LIN {X 0,Y 292.683,Z 375.418,A -85,B 0,C 180,E1 -16601.198,E2 -16601.198} C_VEL
LIN {X 0,Y 293.911,Z 381.437,A -85,B 0,C 180,E1 -16604.861,E2 -16604.861} C_VEL
LIN {X 0,Y 294.978,Z 387.221,A -85,B 0,C 180,E1 -16608.157,E2 -16608.157} C_VEL
LIN {X 0,Y 295.925,Z 392.366,A -85,B 0,C 180,E1 -16610.924,E2 -16610.924} C_VEL
LIN {X 0,Y 296.024,Z 394.252,A -85,B 0,C 180,E1 -16611.884,E2 -16611.884} C_VEL
LIN {X 0,Y 294.406,Z 402.717,A -85,B 0,C 180,E1 -16615.877,E2 -16615.877} C_VEL
LIN {X 0,Y 292.727,Z 412.806,A -85,B 0,C 180,E1 -16620.517,E2 -16620.517} C_VEL
LIN {X 0,Y 291.994,Z 418.301,A -85,B 0,C 180,E1 -16622.943,E2 -16622.943} C_VEL
LIN {X 0,Y 294.998,Z 432.417,A -85,B 0,C 180,E1 -16623.88,E2 -16623.88} C_VEL
LIN {X 0,Y 296.907,Z 445.168,A -85,B 0,C 180,E1 -16624.923,E2 -16624.923} C_VEL
LIN {X 0,Y 297.945,Z 457.115,A -85,B 0,C 180,E1 -16626.095,E2 -16626.095} C_VEL
LIN {X 0,Y 298.202,Z 467.604,A -85,B 0,C 180,E1 -16627.301,E2 -16627.301} C_VEL
LIN {X 0,Y 297.752,Z 476.948,A -85,B 0,C 180,E1 -16628.541,E2 -16628.541} C_VEL
LIN {X 0,Y 296.927,Z 484.846,A -85,B 0,C 180,E1 -16629.748,E2 -16629.748} C_VEL
LIN {X 0,Y 294.74,Z 495.018,A -85,B 0,C 180,E1 -16631.583,E2 -16631.583} C_VEL
LIN {X 0,Y 292.887,Z 504.329,A -85,B 0,C 180,E1 -16633.704,E2 -16633.704} C_VEL
LIN {X 0,Y 291.885,Z 510.195,A -85,B 0,C 180,E1 -16635.357,E2 -16635.357} C_VEL
LIN {X 0,Y 290.834,Z 516.302,A -85,B 0,C 180,E1 -16637.44,E2 -16637.44} C_VEL
LIN {X 0,Y 290.21,Z 521.185,A -85,B 0,C 180,E1 -16639.536,E2 -16639.536} C_VEL
LIN {X 0,Y 290.014,Z 524.981,A -85,B 0,C 180,E1 -16641.641,E2 -16641.641} C_VEL
LIN {X 0,Y 290.054,Z 527.419,A -85,B 0,C 180,E1 -16643.428,E2 -16643.428} C_VEL
LIN {X 0,Y 290.356,Z 529.624,A -85,B 0,C 180,E1 -16645.837,E2 -16645.837} C_VEL
LIN {X 0,Y 290.572,Z 530.346,A -85,B 0,C 180,E1 -16647.228,E2 -16647.228} C_VEL
LIN {X 0,Y 290.579,Z 530.64,A -85,B 0,C 180,E1 -16648.615,E2 -16648.615} C_VEL
LIN {X 0,Y 290.692,Z 530.5,A -85,B 0,C 180,E1 -16650.001,E2 -16650.001} C_VEL
LIN {X 0,Y 290.641,Z 529.922,A -85,B 0,C 180,E1 -16651.387,E2 -16651.387} C_VEL
LIN {X 0,Y 290.644,Z 528.943,A -85,B 0,C 180,E1 -16652.773,E2 -16652.773} C_VEL
LIN {X 0,Y 290.521,Z 527.528,A -85,B 0,C 180,E1 -16654.163,E2 -16654.163} C_VEL
LIN {X 0,Y 290.267,Z 524.115,A -85,B 0,C 180,E1 -16656.483,E2 -16656.483} C_VEL
LIN {X 0,Y 290.179,Z 518.756,A -85,B 0,C 180,E1 -16659.059,E2 -16659.059} C_VEL
LIN {X 0,Y 290.446,Z 513.057,A -85,B 0,C 180,E1 -16661.163,E2 -16661.163} C_VEL
LIN {X 0,Y 291.073,Z 505.963,A -85,B 0,C 180,E1 -16663.262,E2 -16663.262} C_VEL
LIN {X 0,Y 291.825,Z 498.722,A -85,B 0,C 180,E1 -16665.005,E2 -16665.005} C_VEL
LIN {X 0,Y 293.098,Z 490.037,A -85,B 0,C 180,E1 -16666.724,E2 -16666.724} C_VEL
LIN {X 0,Y 294.416,Z 479.281,A -85,B 0,C 180,E1 -16668.44,E2 -16668.44} C_VEL
LIN {X 0,Y 294.522,Z 468.382,A -85,B 0,C 180,E1 -16669.88,E2 -16669.88} C_VEL
LIN {X 0,Y 294.174,Z 456.178,A -85,B 0,C 180,E1 -16671.185,E2 -16671.185} C_VEL
LIN {X 0,Y 293.492,Z 443.337,A -85,B 0,C 180,E1 -16672.251,E2 -16672.251} C_VEL
LIN {X 0,Y 292.3,Z 430.929,A -85,B 0,C 180,E1 -16673.044,E2 -16673.044} C_VEL
LIN {X 0,Y 290.807,Z 419.868,A -85,B 0,C 180,E1 -16673.595,E2 -16673.595} C_VEL
LIN {X 0,Y 291.778,Z 409.748,A -85,B 0,C 180,E1 -16678.015,E2 -16678.015} C_VEL
LIN {X 0,Y 292.997,Z 399.803,A -85,B 0,C 180,E1 -16682.41,E2 -16682.41} C_VEL
LIN {X 0,Y 294.364,Z 390.354,A -85,B 0,C 180,E1 -16686.648,E2 -16686.648} C_VEL
LIN {X 0,Y 294.622,Z 386.771,A -85,B 0,C 180,E1 -16688.333,E2 -16688.333} C_VEL
LIN {X 0,Y 293.697,Z 381.163,A -85,B 0,C 180,E1 -16691.126,E2 -16691.126} C_VEL
LIN {X 0,Y 292.259,Z 373.892,A -85,B 0,C 180,E1 -16694.951,E2 -16694.951} C_VEL
LIN {X 0,Y 291.394,Z 369.189,A -85,B 0,C 180,E1 -16697.647,E2 -16697.647} C_VEL
LIN {X 0,Y 291.357,Z 369.195,A -85,B 0,C 180,E1 -16701.159,E2 -16701.159} C_VEL
LIN {X 0,Y 291.365,Z 369.194,A -85,B 0,C 180,E1 -16704.627,E2 -16704.627} C_VEL
LIN {X 0,Y 291.375,Z 369.189,A -85,B 0,C 180,E1 -16707.951,E2 -16707.951} C_VEL
LIN {X 0,Y 291.382,Z 369.189,A -85,B 0,C 180,E1 -16711.158,E2 -16711.158} C_VEL
LIN {X 0,Y 291.417,Z 369.185,A -85,B 0,C 180,E1 -16714.272,E2 -16714.272} C_VEL
LIN {X 0,Y 291.387,Z 369.188,A -85,B 0,C 180,E1 -16717.3,E2 -16717.3} C_VEL
LIN {X 0,Y 291.463,Z 369.181,A -85,B 0,C 180,E1 -16720.271,E2 -16720.271} C_VEL
LIN {X 0,Y 291.56,Z 369.169,A -85,B 0,C 180,E1 -16724.624,E2 -16724.624} C_VEL
LIN {X 0,Y 291.542,Z 369.169,A -85,B 0,C 180,E1 -16728.881,E2 -16728.881} C_VEL
LIN {X 0,Y 291.716,Z 369.146,A -85,B 0,C 180,E1 -16731.689,E2 -16731.689} C_VEL
LIN {X 0,Y 291.636,Z 369.159,A -85,B 0,C 180,E1 -16734.469,E2 -16734.469} C_VEL
LIN {X 0,Y 291.895,Z 369.121,A -85,B 0,C 180,E1 -16738.621,E2 -16738.621} C_VEL
LIN {X 0,Y 291.896,Z 369.122,A -85,B 0,C 180,E1 -16741.38,E2 -16741.38} C_VEL
LIN {X 0,Y 291.753,Z 369.136,A -85,B 0,C 180,E1 -16746.918,E2 -16746.918} C_VEL
LIN {X 0,Y 291.635,Z 369.156,A -85,B 0,C 180,E1 -16749.712,E2 -16749.712} C_VEL
LIN {X 0,Y 291.528,Z 369.169,A -85,B 0,C 180,E1 -16753.95,E2 -16753.95} C_VEL
LIN {X 0,Y 291.493,Z 369.171,A -85,B 0,C 180,E1 -16756.818,E2 -16756.818} C_VEL
LIN {X 0,Y 291.457,Z 369.181,A -85,B 0,C 180,E1 -16759.875,E2 -16759.875} C_VEL
LIN {X 0,Y 291.407,Z 369.184,A -85,B 0,C 180,E1 -16764.205,E2 -16764.205} C_VEL
LIN {X 0,Y 291.427,Z 369.183,A -85,B 0,C 180,E1 -16767.272,E2 -16767.272} C_VEL
LIN {X 0,Y 291.343,Z 369.188,A -85,B 0,C 180,E1 -16770.437,E2 -16770.437} C_VEL
LIN {X 0,Y 291.351,Z 369.194,A -85,B 0,C 180,E1 -16773.698,E2 -16773.698} C_VEL
LIN {X 0,Y 291.401,Z 369.187,A -85,B 0,C 180,E1 -16777.259,E2 -16777.259} C_VEL
LIN {X 0,Y 291.341,Z 369.192,A -85,B 0,C 180,E1 -16780.642,E2 -16780.642} C_VEL
LIN {X 0,Y 291.32,Z 369.193,A -85,B 0,C 180,E1 -16784.397,E2 -16784.397} C_VEL
LIN {X 0,Y 291.333,Z 369.192,A -85,B 0,C 180,E1 -16788.404,E2 -16788.404} C_VEL
LIN {X 0,Y 291.359,Z 369.193,A -85,B 0,C 180,E1 -16791.158,E2 -16791.158} C_VEL
LIN {X 0,Y 291.367,Z 369.189,A -85,B 0,C 180,E1 -16794.626,E2 -16794.626} C_VEL
LIN {X 0,Y 291.378,Z 369.187,A -85,B 0,C 180,E1 -16797.95,E2 -16797.95} C_VEL
LIN {X 0,Y 291.389,Z 369.19,A -85,B 0,C 180,E1 -16801.158,E2 -16801.158} C_VEL
LIN {X 0,Y 291.423,Z 369.183,A -85,B 0,C 180,E1 -16804.271,E2 -16804.271} C_VEL
LIN {X 0,Y 291.388,Z 369.189,A -85,B 0,C 180,E1 -16807.299,E2 -16807.299} C_VEL
LIN {X 0,Y 291.464,Z 369.178,A -85,B 0,C 180,E1 -16810.27,E2 -16810.27} C_VEL
LIN {X 0,Y 291.563,Z 369.169,A -85,B 0,C 180,E1 -16814.837,E2 -16814.837} C_VEL
LIN {X 0,Y 291.568,Z 369.167,A -85,B 0,C 180,E1 -16815.316,E2 -16815.316} C_VEL
LIN {X 0,Y 295.833,Z 381.993,A -85,B 0,C 180,E1 -16816.562,E2 -16816.562} C_VEL
LIN {X 0,Y 298.818,Z 392.412,A -85,B 0,C 180,E1 -16817.779,E2 -16817.779} C_VEL
LIN {X 0,Y 299.175,Z 393.845,A -85,B 0,C 180,E1 -16817.965,E2 -16817.965} C_VEL
LIN {X 0,Y 298.005,Z 405.109,A -85,B 0,C 180,E1 -16819.296,E2 -16819.296} C_VEL
LIN {X 0,Y 296.886,Z 415.247,A -85,B 0,C 180,E1 -16820.804,E2 -16820.804} C_VEL
LIN {X 0,Y 295.741,Z 424.376,A -85,B 0,C 180,E1 -16822.489,E2 -16822.489} C_VEL
LIN {X 0,Y 294.418,Z 433.245,A -85,B 0,C 180,E1 -16824.52,E2 -16824.52} C_VEL
LIN {X 0,Y 293.334,Z 440.396,A -85,B 0,C 180,E1 -16826.565,E2 -16826.565} C_VEL
LIN {X 0,Y 292.496,Z 446.124,A -85,B 0,C 180,E1 -16828.622,E2 -16828.622} C_VEL
LIN {X 0,Y 291.905,Z 450.636,A -85,B 0,C 180,E1 -16830.689,E2 -16830.689} C_VEL
LIN {X 0,Y 291.33,Z 454.107,A -85,B 0,C 180,E1 -16832.764,E2 -16832.764} C_VEL
LIN {X 0,Y 291.196,Z 455.839,A -85,B 0,C 180,E1 -16834.151,E2 -16834.151} C_VEL
LIN {X 0,Y 291.213,Z 457.151,A -85,B 0,C 180,E1 -16835.539,E2 -16835.539} C_VEL
LIN {X 0,Y 291.178,Z 458.652,A -85,B 0,C 180,E1 -16838.269,E2 -16838.269} C_VEL
LIN {X 0,Y 291.268,Z 458.81,A -85,B 0,C 180,E1 -16839.723,E2 -16839.723} C_VEL
LIN {X 0,Y 291.675,Z 457.948,A -85,B 0,C 180,E1 -16842.523,E2 -16842.523} C_VEL
LIN {X 0,Y 292.039,Z 456.928,A -85,B 0,C 180,E1 -16843.924,E2 -16843.924} C_VEL
LIN {X 0,Y 292.98,Z 454.095,A -85,B 0,C 180,E1 -16846.356,E2 -16846.356} C_VEL
LIN {X 0,Y 294.179,Z 449.853,A -85,B 0,C 180,E1 -16848.814,E2 -16848.814} C_VEL
LIN {X 0,Y 295.431,Z 445.004,A -85,B 0,C 180,E1 -16850.905,E2 -16850.905} C_VEL
LIN {X 0,Y 296.905,Z 439.068,A -85,B 0,C 180,E1 -16852.915,E2 -16852.915} C_VEL
LIN {X 0,Y 298.493,Z 432.492,A -85,B 0,C 180,E1 -16854.702,E2 -16854.702} C_VEL
LIN {X 0,Y 300.367,Z 423.575,A -85,B 0,C 180,E1 -16856.659,E2 -16856.659} C_VEL
LIN {X 0,Y 302.222,Z 413.214,A -85,B 0,C 180,E1 -16858.47,E2 -16858.47} C_VEL
LIN {X 0,Y 303.808,Z 403.47,A -85,B 0,C 180,E1 -16859.825,E2 -16859.825} C_VEL
LIN {X 0,Y 303.684,Z 401.365,A -85,B 0,C 180,E1 -16860.122,E2 -16860.122} C_VEL
LIN {X 0,Y 300.573,Z 391.397,A -85,B 0,C 180,E1 -16861.672,E2 -16861.672} C_VEL
LIN {X 0,Y 296.215,Z 380.226,A -85,B 0,C 180,E1 -16863.243,E2 -16863.243} C_VEL
LIN {X 0,Y 292.253,Z 371.834,A -85,B 0,C 180,E1 -16864.331,E2 -16864.331} C_VEL
LIN {X 0,Y 291.371,Z 369.192,A -85,B 0,C 180,E1 -16864.659,E2 -16864.659} C_VEL
LIN {X 0,Y 291.376,Z 369.194,A -85,B 0,C 180,E1 -16867.253,E2 -16867.253} C_VEL
LIN {X 0,Y 291.332,Z 369.197,A -85,B 0,C 180,E1 -16870.641,E2 -16870.641} C_VEL
LIN {X 0,Y 291.288,Z 369.2,A -85,B 0,C 180,E1 -16874.401,E2 -16874.401} C_VEL
LIN {X 0,Y 291.354,Z 369.197,A -85,B 0,C 180,E1 -16878.397,E2 -16878.397} C_VEL
LIN {X 0,Y 291.379,Z 369.192,A -85,B 0,C 180,E1 -16881.162,E2 -16881.162} C_VEL
LIN {X 0,Y 291.384,Z 369.188,A -85,B 0,C 180,E1 -16884.629,E2 -16884.629} C_VEL
LIN {X 0,Y 291.373,Z 369.173,A -85,B 0,C 180,E1 -16887.95,E2 -16887.95} C_VEL
LIN {X 0,Y 291.38,Z 369.158,A -85,B 0,C 180,E1 -16891.158,E2 -16891.158} C_VEL
LIN {X 0,Y 291.414,Z 369.185,A -85,B 0,C 180,E1 -16894.271,E2 -16894.271} C_VEL
LIN {X 0,Y 291.379,Z 369.178,A -85,B 0,C 180,E1 -16897.299,E2 -16897.299} C_VEL
LIN {X 0,Y 291.455,Z 369.179,A -85,B 0,C 180,E1 -16900.27,E2 -16900.27} C_VEL
LIN {X 0,Y 291.551,Z 369.17,A -85,B 0,C 180,E1 -16904.623,E2 -16904.623} C_VEL
LIN {X 0,Y 291.535,Z 369.171,A -85,B 0,C 180,E1 -16908.88,E2 -16908.88} C_VEL
LIN {X 0,Y 291.705,Z 369.15,A -85,B 0,C 180,E1 -16911.688,E2 -16911.688} C_VEL
LIN {X 0,Y 291.603,Z 369.148,A -85,B 0,C 180,E1 -16914.707,E2 -16914.707} C_VEL
LIN {X 0,Y 291.89,Z 369.123,A -85,B 0,C 180,E1 -16918.62,E2 -16918.62} C_VEL
LIN {X 0,Y 291.91,Z 369.114,A -85,B 0,C 180,E1 -16920.74,E2 -16920.74} C_VEL
LIN {X 0,Y 291.165,Z 369.216,A -85,B 0,C 180,E1 -16921.888,E2 -16921.888} C_VEL
LIN {X 0,Y 288.167,Z 369.588,A -85,B 0,C 180,E1 -16923.754,E2 -16923.754} C_VEL
LIN {X 0,Y 285.7,Z 369.889,A -85,B 0,C 180,E1 -16925.27,E2 -16925.27} C_VEL
LIN {X 0,Y 284.71,Z 370.017,A -85,B 0,C 180,E1 -16926.448,E2 -16926.448} C_VEL
LIN {X 0,Y 284.666,Z 370.023,A -85,B 0,C 180,E1 -16926.846,E2 -16926.846} C_VEL
LIN {X 0,Y 284.562,Z 370.029,A -85,B 0,C 180,E1 -16929.955,E2 -16929.955} C_VEL
LIN {X 0,Y 284.477,Z 370.042,A -85,B 0,C 180,E1 -16934.303,E2 -16934.303} C_VEL
LIN {X 0,Y 284.421,Z 370.051,A -85,B 0,C 180,E1 -16937.248,E2 -16937.248} C_VEL
LIN {X 0,Y 284.374,Z 370.06,A -85,B 0,C 180,E1 -16940.242,E2 -16940.242} C_VEL
LIN {X 0,Y 284.365,Z 370.061,A -85,B 0,C 180,E1 -16943.876,E2 -16943.876} C_VEL
LIN {X 0,Y 284.393,Z 370.064,A -85,B 0,C 180,E1 -16947.174,E2 -16947.174} C_VEL
LIN {X 0,Y 284.292,Z 370.076,A -85,B 0,C 180,E1 -16951.275,E2 -16951.275} C_VEL
LIN {X 0,Y 284.345,Z 370.064,A -85,B 0,C 180,E1 -16955.803,E2 -16955.803} C_VEL
LIN {X 0,Y 284.38,Z 370.218,A -85,B 0,C 180,E1 -16956.379,E2 -16956.379} C_VEL
LIN {X 0,Y 285.532,Z 375.84,A -85,B 0,C 180,E1 -16960.27,E2 -16960.27} C_VEL
LIN {X 0,Y 286.736,Z 381.797,A -85,B 0,C 180,E1 -16964.061,E2 -16964.061} C_VEL
LIN {X 0,Y 288,Z 388.459,A -85,B 0,C 180,E1 -16967.97,E2 -16967.97} C_VEL
LIN {X 0,Y 289,Z 394.136,A -85,B 0,C 180,E1 -16971.095,E2 -16971.095} C_VEL
LIN {X 0,Y 288.762,Z 396.965,A -85,B 0,C 180,E1 -16972.523,E2 -16972.523} C_VEL
LIN {X 0,Y 286.964,Z 405.919,A -85,B 0,C 180,E1 -16976.845,E2 -16976.845} C_VEL
LIN {X 0,Y 285.399,Z 415.403,A -85,B 0,C 180,E1 -16981.303,E2 -16981.303} C_VEL
LIN {X 0,Y 285.143,Z 417.2,A -85,B 0,C 180,E1 -16982.13,E2 -16982.13} C_VEL
LIN {X 0,Y 287.856,Z 429.507,A -85,B 0,C 180,E1 -16982.975,E2 -16982.975} C_VEL
LIN {X 0,Y 289.99,Z 442.581,A -85,B 0,C 180,E1 -16984.06,E2 -16984.06} C_VEL
LIN {X 0,Y 291.121,Z 454.499,A -85,B 0,C 180,E1 -16985.231,E2 -16985.231} C_VEL
LIN {X 0,Y 291.522,Z 466.194,A -85,B 0,C 180,E1 -16986.6,E2 -16986.6} C_VEL
LIN {X 0,Y 291.067,Z 476.581,A -85,B 0,C 180,E1 -16988.023,E2 -16988.023} C_VEL
LIN {X 0,Y 290.038,Z 485.402,A -85,B 0,C 180,E1 -16989.431,E2 -16989.431} C_VEL
LIN {X 0,Y 287.993,Z 494.494,A -85,B 0,C 180,E1 -16991.136,E2 -16991.136} C_VEL
LIN {X 0,Y 286.038,Z 503.818,A -85,B 0,C 180,E1 -16993.324,E2 -16993.324} C_VEL
LIN {X 0,Y 284.721,Z 510.666,A -85,B 0,C 180,E1 -16995.345,E2 -16995.345} C_VEL
LIN {X 0,Y 283.581,Z 517.334,A -85,B 0,C 180,E1 -16997.84,E2 -16997.84} C_VEL
LIN {X 0,Y 283.059,Z 521.803,A -85,B 0,C 180,E1 -16999.992,E2 -16999.992} C_VEL
LIN {X 0,Y 282.934,Z 524.207,A -85,B 0,C 180,E1 -17001.43,E2 -17001.43} C_VEL
LIN {X 0,Y 282.99,Z 526.775,A -85,B 0,C 180,E1 -17003.409,E2 -17003.409} C_VEL
LIN {X 0,Y 283.275,Z 528.786,A -85,B 0,C 180,E1 -17005.733,E2 -17005.733} C_VEL
LIN {X 0,Y 283.52,Z 529.496,A -85,B 0,C 180,E1 -17007.159,E2 -17007.159} C_VEL
LIN {X 0,Y 283.531,Z 529.768,A -85,B 0,C 180,E1 -17008.581,E2 -17008.581} C_VEL
LIN {X 0,Y 283.647,Z 529.602,A -85,B 0,C 180,E1 -17010.001,E2 -17010.001} C_VEL
LIN {X 0,Y 283.593,Z 529.007,A -85,B 0,C 180,E1 -17011.421,E2 -17011.421} C_VEL
LIN {X 0,Y 283.596,Z 528.01,A -85,B 0,C 180,E1 -17012.842,E2 -17012.842} C_VEL
LIN {X 0,Y 283.455,Z 526.566,A -85,B 0,C 180,E1 -17014.267,E2 -17014.267} C_VEL
LIN {X 0,Y 283.181,Z 522.613,A -85,B 0,C 180,E1 -17016.917,E2 -17016.917} C_VEL
LIN {X 0,Y 283.108,Z 517.697,A -85,B 0,C 180,E1 -17019.287,E2 -17019.287} C_VEL
LIN {X 0,Y 283.414,Z 511.954,A -85,B 0,C 180,E1 -17021.443,E2 -17021.443} C_VEL
LIN {X 0,Y 284.098,Z 504.802,A -85,B 0,C 180,E1 -17023.593,E2 -17023.593} C_VEL
LIN {X 0,Y 284.849,Z 497.495,A -85,B 0,C 180,E1 -17025.382,E2 -17025.382} C_VEL
LIN {X 0,Y 286.409,Z 487.741,A -85,B 0,C 180,E1 -17027.31,E2 -17027.31} C_VEL
LIN {X 0,Y 287.492,Z 477.857,A -85,B 0,C 180,E1 -17028.9,E2 -17028.9} C_VEL
LIN {X 0,Y 287.492,Z 466.799,A -85,B 0,C 180,E1 -17030.388,E2 -17030.388} C_VEL
LIN {X 0,Y 287.242,Z 454.552,A -85,B 0,C 180,E1 -17031.702,E2 -17031.702} C_VEL
LIN {X 0,Y 286.492,Z 441.166,A -85,B 0,C 180,E1 -17032.825,E2 -17032.825} C_VEL
LIN {X 0,Y 285.104,Z 428.095,A -85,B 0,C 180,E1 -17033.66,E2 -17033.66} C_VEL
LIN {X 0,Y 283.82,Z 419.071,A -85,B 0,C 180,E1 -17034.101,E2 -17034.101} C_VEL
LIN {X 0,Y 284.864,Z 408.71,A -85,B 0,C 180,E1 -17038.758,E2 -17038.758} C_VEL
LIN {X 0,Y 286.02,Z 399.96,A -85,B 0,C 180,E1 -17042.724,E2 -17042.724} C_VEL
LIN {X 0,Y 287.363,Z 391.118,A -85,B 0,C 180,E1 -17046.82,E2 -17046.82} C_VEL
LIN {X 0,Y 287.573,Z 387.519,A -85,B 0,C 180,E1 -17048.551,E2 -17048.551} C_VEL
LIN {X 0,Y 286.398,Z 380.811,A -85,B 0,C 180,E1 -17052.007,E2 -17052.007} C_VEL
LIN {X 0,Y 284.901,Z 372.942,A -85,B 0,C 180,E1 -17056.314,E2 -17056.314} C_VEL
LIN {X 0,Y 284.329,Z 370.069,A -85,B 0,C 180,E1 -17058.057,E2 -17058.057} C_VEL
LIN {X 0,Y 284.326,Z 370.069,A -85,B 0,C 180,E1 -17062.279,E2 -17062.279} C_VEL
LIN {X 0,Y 284.313,Z 370.071,A -85,B 0,C 180,E1 -17065.351,E2 -17065.351} C_VEL
LIN {X 0,Y 284.298,Z 370.073,A -85,B 0,C 180,E1 -17068.726,E2 -17068.726} C_VEL
LIN {X 0,Y 284.399,Z 370.061,A -85,B 0,C 180,E1 -17072.828,E2 -17072.828} C_VEL
LIN {X 0,Y 284.372,Z 370.066,A -85,B 0,C 180,E1 -17076.708,E2 -17076.708} C_VEL
LIN {X 0,Y 284.409,Z 370.058,A -85,B 0,C 180,E1 -17081.262,E2 -17081.262} C_VEL
LIN {X 0,Y 284.498,Z 370.05,A -85,B 0,C 180,E1 -17084.46,E2 -17084.46} C_VEL
LIN {X 0,Y 284.494,Z 370.049,A -85,B 0,C 180,E1 -17088.602,E2 -17088.602} C_VEL
LIN {X 0,Y 284.666,Z 370.024,A -85,B 0,C 180,E1 -17091.482,E2 -17091.482} C_VEL
LIN {X 0,Y 284.607,Z 370.036,A -85,B 0,C 180,E1 -17094.332,E2 -17094.332} C_VEL
LIN {X 0,Y 284.861,Z 369.997,A -85,B 0,C 180,E1 -17098.587,E2 -17098.587} C_VEL
LIN {X 0,Y 284.862,Z 369.998,A -85,B 0,C 180,E1 -17101.414,E2 -17101.414} C_VEL
LIN {X 0,Y 284.705,Z 370.013,A -85,B 0,C 180,E1 -17107.09,E2 -17107.09} C_VEL
LIN {X 0,Y 284.573,Z 370.038,A -85,B 0,C 180,E1 -17109.956,E2 -17109.956} C_VEL
LIN {X 0,Y 284.488,Z 370.042,A -85,B 0,C 180,E1 -17114.303,E2 -17114.303} C_VEL
LIN {X 0,Y 284.432,Z 370.051,A -85,B 0,C 180,E1 -17117.248,E2 -17117.248} C_VEL
LIN {X 0,Y 284.386,Z 370.059,A -85,B 0,C 180,E1 -17120.242,E2 -17120.242} C_VEL
LIN {X 0,Y 284.376,Z 370.06,A -85,B 0,C 180,E1 -17123.875,E2 -17123.875} C_VEL
LIN {X 0,Y 284.402,Z 370.057,A -85,B 0,C 180,E1 -17127.173,E2 -17127.173} C_VEL
LIN {X 0,Y 284.302,Z 370.067,A -85,B 0,C 180,E1 -17131.274,E2 -17131.274} C_VEL
LIN {X 0,Y 284.368,Z 370.064,A -85,B 0,C 180,E1 -17135.354,E2 -17135.354} C_VEL
LIN {X 0,Y 284.329,Z 370.065,A -85,B 0,C 180,E1 -17138.167,E2 -17138.167} C_VEL
LIN {X 0,Y 284.275,Z 370.071,A -85,B 0,C 180,E1 -17142.124,E2 -17142.124} C_VEL
LIN {X 0,Y 284.274,Z 370.071,A -85,B 0,C 180,E1 -17146.192,E2 -17146.192} C_VEL
LIN {X 0,Y 284.312,Z 370.066,A -85,B 0,C 180,E1 -17150.024,E2 -17150.024} C_VEL
LIN {X 0,Y 284.338,Z 370.065,A -85,B 0,C 180,E1 -17153.614,E2 -17153.614} C_VEL
LIN {X 0,Y 284.314,Z 370.071,A -85,B 0,C 180,E1 -17157.189,E2 -17157.189} C_VEL
LIN {X 0,Y 284.365,Z 370.062,A -85,B 0,C 180,E1 -17160.376,E2 -17160.376} C_VEL
LIN {X 0,Y 284.384,Z 370.06,A -85,B 0,C 180,E1 -17163.586,E2 -17163.586} C_VEL
LIN {X 0,Y 284.373,Z 370.063,A -85,B 0,C 180,E1 -17166.706,E2 -17166.706} C_VEL
LIN {X 0,Y 284.41,Z 370.059,A -85,B 0,C 180,E1 -17171.261,E2 -17171.261} C_VEL
LIN {X 0,Y 284.543,Z 370.186,A -85,B 0,C 180,E1 -17174.821,E2 -17174.821} C_VEL
LIN {X 0,Y 288.815,Z 382.8,A -85,B 0,C 180,E1 -17176.09,E2 -17176.09} C_VEL
LIN {X 0,Y 291.742,Z 392.861,A -85,B 0,C 180,E1 -17177.3,E2 -17177.3} C_VEL
LIN {X 0,Y 292.372,Z 395.773,A -85,B 0,C 180,E1 -17177.681,E2 -17177.681} C_VEL
LIN {X 0,Y 291.132,Z 406.849,A -85,B 0,C 180,E1 -17179.04,E2 -17179.04} C_VEL
LIN {X 0,Y 289.982,Z 416.81,A -85,B 0,C 180,E1 -17180.583,E2 -17180.583} C_VEL
LIN {X 0,Y 288.793,Z 425.792,A -85,B 0,C 180,E1 -17182.307,E2 -17182.307} C_VEL
LIN {X 0,Y 287.426,Z 434.571,A -85,B 0,C 180,E1 -17184.386,E2 -17184.386} C_VEL
LIN {X 0,Y 286.316,Z 441.641,A -85,B 0,C 180,E1 -17186.481,E2 -17186.481} C_VEL
LIN {X 0,Y 285.463,Z 447.282,A -85,B 0,C 180,E1 -17188.588,E2 -17188.588} C_VEL
LIN {X 0,Y 284.859,Z 451.727,A -85,B 0,C 180,E1 -17190.706,E2 -17190.706} C_VEL
LIN {X 0,Y 284.272,Z 455.146,A -85,B 0,C 180,E1 -17192.833,E2 -17192.833} C_VEL
LIN {X 0,Y 284.157,Z 458.121,A -85,B 0,C 180,E1 -17195.677,E2 -17195.677} C_VEL
LIN {X 0,Y 284.146,Z 459.529,A -85,B 0,C 180,E1 -17198.365,E2 -17198.365} C_VEL
LIN {X 0,Y 284.256,Z 459.674,A -85,B 0,C 180,E1 -17199.965,E2 -17199.965} C_VEL
LIN {X 0,Y 284.715,Z 458.759,A -85,B 0,C 180,E1 -17202.835,E2 -17202.835} C_VEL
LIN {X 0,Y 285.109,Z 457.687,A -85,B 0,C 180,E1 -17204.27,E2 -17204.27} C_VEL
LIN {X 0,Y 286.057,Z 454.984,A -85,B 0,C 180,E1 -17206.628,E2 -17206.628} C_VEL
LIN {X 0,Y 287.401,Z 450.491,A -85,B 0,C 180,E1 -17209.275,E2 -17209.275} C_VEL
LIN {X 0,Y 288.743,Z 445.575,A -85,B 0,C 180,E1 -17211.413,E2 -17211.413} C_VEL
LIN {X 0,Y 290.322,Z 439.561,A -85,B 0,C 180,E1 -17213.466,E2 -17213.466} C_VEL
LIN {X 0,Y 292.307,Z 431.428,A -85,B 0,C 180,E1 -17215.643,E2 -17215.643} C_VEL
LIN {X 0,Y 294.169,Z 422.87,A -85,B 0,C 180,E1 -17217.476,E2 -17217.476} C_VEL
LIN {X 0,Y 295.925,Z 413.351,A -85,B 0,C 180,E1 -17219.133,E2 -17219.133} C_VEL
LIN {X 0,Y 297.285,Z 405.45,A -85,B 0,C 180,E1 -17220.247,E2 -17220.247} C_VEL
LIN {X 0,Y 297.101,Z 402.931,A -85,B 0,C 180,E1 -17220.631,E2 -17220.631} C_VEL
LIN {X 0,Y 293.658,Z 392.367,A -85,B 0,C 180,E1 -17222.355,E2 -17222.355} C_VEL
LIN {X 0,Y 289.363,Z 381.424,A -85,B 0,C 180,E1 -17223.959,E2 -17223.959} C_VEL
LIN {X 0,Y 285.305,Z 372.882,A -85,B 0,C 180,E1 -17225.12,E2 -17225.12} C_VEL
LIN {X 0,Y 284.331,Z 370.073,A -85,B 0,C 180,E1 -17225.456,E2 -17225.456} C_VEL
LIN {X 0,Y 284.312,Z 370.07,A -85,B 0,C 180,E1 -17228.168,E2 -17228.168} C_VEL
LIN {X 0,Y 284.268,Z 370.074,A -85,B 0,C 180,E1 -17232.123,E2 -17232.123} C_VEL
LIN {X 0,Y 284.271,Z 370.077,A -85,B 0,C 180,E1 -17236.191,E2 -17236.191} C_VEL
LIN {X 0,Y 284.35,Z 370.063,A -85,B 0,C 180,E1 -17240.012,E2 -17240.012} C_VEL
LIN {X 0,Y 284.353,Z 370.06,A -85,B 0,C 180,E1 -17243.617,E2 -17243.617} C_VEL
LIN {X 0,Y 284.307,Z 370.063,A -85,B 0,C 180,E1 -17247.188,E2 -17247.188} C_VEL
LIN {X 0,Y 284.357,Z 370.025,A -85,B 0,C 180,E1 -17250.375,E2 -17250.375} C_VEL
LIN {X 0,Y 284.375,Z 370.059,A -85,B 0,C 180,E1 -17253.586,E2 -17253.586} C_VEL
LIN {X 0,Y 284.363,Z 370.051,A -85,B 0,C 180,E1 -17256.706,E2 -17256.706} C_VEL
LIN {X 0,Y 284.401,Z 370.052,A -85,B 0,C 180,E1 -17261.261,E2 -17261.261} C_VEL
LIN {X 0,Y 284.489,Z 370.049,A -85,B 0,C 180,E1 -17264.458,E2 -17264.458} C_VEL
LIN {X 0,Y 284.487,Z 370.049,A -85,B 0,C 180,E1 -17268.601,E2 -17268.601} C_VEL
LIN {X 0,Y 284.656,Z 370.028,A -85,B 0,C 180,E1 -17271.481,E2 -17271.481} C_VEL
LIN {X 0,Y 284.599,Z 370.02,A -85,B 0,C 180,E1 -17274.331,E2 -17274.331} C_VEL
LIN {X 0,Y 284.856,Z 369.999,A -85,B 0,C 180,E1 -17278.586,E2 -17278.586} C_VEL
LIN {X 0,Y 284.856,Z 369.999,A -85,B 0,C 180,E1 -17281.413,E2 -17281.413} C_VEL
LIN {X 0,Y 284.666,Z 370.023,A -85,B 0,C 180,E1 -17286.846,E2 -17286.846} C_VEL
LIN {X 0,Y 284.057,Z 370.107,A -85,B 0,C 180,E1 -17288.026,E2 -17288.026} C_VEL
LIN {X 0,Y 281.098,Z 370.474,A -85,B 0,C 180,E1 -17289.942,E2 -17289.942} C_VEL
LIN {X 0,Y 278.55,Z 370.787,A -85,B 0,C 180,E1 -17291.5,E2 -17291.5} C_VEL
LIN {X 0,Y 277.48,Z 370.92,A -85,B 0,C 180,E1 -17292.711,E2 -17292.711} C_VEL
LIN {X 0,Y 277.41,Z 370.924,A -85,B 0,C 180,E1 -17293.122,E2 -17293.122} C_VEL
LIN {X 0,Y 277.402,Z 370.931,A -85,B 0,C 180,E1 -17296.182,E2 -17296.182} C_VEL
LIN {X 0,Y 277.341,Z 370.935,A -85,B 0,C 180,E1 -17300.35,E2 -17300.35} C_VEL
LIN {X 0,Y 277.315,Z 370.94,A -85,B 0,C 180,E1 -17304.171,E2 -17304.171} C_VEL
LIN {X 0,Y 277.322,Z 370.945,A -85,B 0,C 180,E1 -17307.506,E2 -17307.506} C_VEL
LIN {X 0,Y 277.268,Z 370.951,A -85,B 0,C 180,E1 -17310.482,E2 -17310.482} C_VEL
LIN {X 0,Y 277.313,Z 370.941,A -85,B 0,C 180,E1 -17315.209,E2 -17315.209} C_VEL
LIN {X 0,Y 277.411,Z 371.459,A -85,B 0,C 180,E1 -17315.838,E2 -17315.838} C_VEL
LIN {X 0,Y 278.625,Z 377.319,A -85,B 0,C 180,E1 -17320.009,E2 -17320.009} C_VEL
LIN {X 0,Y 279.768,Z 383.119,A -85,B 0,C 180,E1 -17323.819,E2 -17323.819} C_VEL
LIN {X 0,Y 280.917,Z 389.221,A -85,B 0,C 180,E1 -17327.509,E2 -17327.509} C_VEL
LIN {X 0,Y 281.911,Z 394.639,A -85,B 0,C 180,E1 -17330.608,E2 -17330.608} C_VEL
LIN {X 0,Y 282.033,Z 396.233,A -85,B 0,C 180,E1 -17331.468,E2 -17331.468} C_VEL
LIN {X 0,Y 280.998,Z 401.291,A -85,B 0,C 180,E1 -17334.004,E2 -17334.004} C_VEL
LIN {X 0,Y 279.392,Z 409.647,A -85,B 0,C 180,E1 -17338.114,E2 -17338.114} C_VEL
LIN {X 0,Y 278.331,Z 416.232,A -85,B 0,C 180,E1 -17341.28,E2 -17341.28} C_VEL
LIN {X 0,Y 281.135,Z 429.112,A -85,B 0,C 180,E1 -17342.204,E2 -17342.204} C_VEL
LIN {X 0,Y 283.236,Z 441.536,A -85,B 0,C 180,E1 -17343.288,E2 -17343.288} C_VEL
LIN {X 0,Y 284.486,Z 454.58,A -85,B 0,C 180,E1 -17344.629,E2 -17344.629} C_VEL
LIN {X 0,Y 284.823,Z 466.832,A -85,B 0,C 180,E1 -17346.136,E2 -17346.136} C_VEL
LIN {X 0,Y 284.267,Z 477.4,A -85,B 0,C 180,E1 -17347.66,E2 -17347.66} C_VEL
LIN {X 0,Y 283.368,Z 484.949,A -85,B 0,C 180,E1 -17348.924,E2 -17348.924} C_VEL
LIN {X 0,Y 281.251,Z 493.969,A -85,B 0,C 180,E1 -17350.666,E2 -17350.666} C_VEL
LIN {X 0,Y 279.237,Z 503.019,A -85,B 0,C 180,E1 -17352.848,E2 -17352.848} C_VEL
LIN {X 0,Y 277.842,Z 510.005,A -85,B 0,C 180,E1 -17354.974,E2 -17354.974} C_VEL
LIN {X 0,Y 276.576,Z 516.623,A -85,B 0,C 180,E1 -17357.527,E2 -17357.527} C_VEL
LIN {X 0,Y 276.007,Z 521.052,A -85,B 0,C 180,E1 -17359.734,E2 -17359.734} C_VEL
LIN {X 0,Y 275.881,Z 523.439,A -85,B 0,C 180,E1 -17361.209,E2 -17361.209} C_VEL
LIN {X 0,Y 275.934,Z 526.118,A -85,B 0,C 180,E1 -17363.376,E2 -17363.376} C_VEL
LIN {X 0,Y 276.197,Z 527.95,A -85,B 0,C 180,E1 -17365.623,E2 -17365.623} C_VEL
LIN {X 0,Y 276.467,Z 528.647,A -85,B 0,C 180,E1 -17367.087,E2 -17367.087} C_VEL
LIN {X 0,Y 276.483,Z 528.889,A -85,B 0,C 180,E1 -17368.544,E2 -17368.544} C_VEL
LIN {X 0,Y 276.602,Z 528.704,A -85,B 0,C 180,E1 -17370.001,E2 -17370.001} C_VEL
LIN {X 0,Y 276.545,Z 528.092,A -85,B 0,C 180,E1 -17371.457,E2 -17371.457} C_VEL
LIN {X 0,Y 276.548,Z 527.077,A -85,B 0,C 180,E1 -17372.914,E2 -17372.914} C_VEL
LIN {X 0,Y 276.39,Z 525.597,A -85,B 0,C 180,E1 -17374.376,E2 -17374.376} C_VEL
LIN {X 0,Y 276.107,Z 521.893,A -85,B 0,C 180,E1 -17376.926,E2 -17376.926} C_VEL
LIN {X 0,Y 276.061,Z 516.639,A -85,B 0,C 180,E1 -17379.526,E2 -17379.526} C_VEL
LIN {X 0,Y 276.393,Z 510.847,A -85,B 0,C 180,E1 -17381.738,E2 -17381.738} C_VEL
LIN {X 0,Y 277.126,Z 503.622,A -85,B 0,C 180,E1 -17383.942,E2 -17383.942} C_VEL
LIN {X 0,Y 278.215,Z 494.596,A -85,B 0,C 180,E1 -17386.134,E2 -17386.134} C_VEL
LIN {X 0,Y 279.5,Z 486.404,A -85,B 0,C 180,E1 -17387.752,E2 -17387.752} C_VEL
LIN {X 0,Y 280.501,Z 477.629,A -85,B 0,C 180,E1 -17389.2,E2 -17389.2} C_VEL
LIN {X 0,Y 280.519,Z 466.905,A -85,B 0,C 180,E1 -17390.7,E2 -17390.7} C_VEL
LIN {X 0,Y 280.327,Z 454.561,A -85,B 0,C 180,E1 -17392.091,E2 -17392.091} C_VEL
LIN {X 0,Y 279.653,Z 441.73,A -85,B 0,C 180,E1 -17393.22,E2 -17393.22} C_VEL
LIN {X 0,Y 278.307,Z 428.481,A -85,B 0,C 180,E1 -17394.12,E2 -17394.12} C_VEL
LIN {X 0,Y 276.834,Z 418.137,A -85,B 0,C 180,E1 -17394.667,E2 -17394.667} C_VEL
LIN {X 0,Y 277.996,Z 407.628,A -85,B 0,C 180,E1 -17399.538,E2 -17399.538} C_VEL
LIN {X 0,Y 279.267,Z 398.454,A -85,B 0,C 180,E1 -17403.853,E2 -17403.853} C_VEL
LIN {X 0,Y 280.366,Z 391.878,A -85,B 0,C 180,E1 -17406.987,E2 -17406.987} C_VEL
LIN {X 0,Y 280.493,Z 388.212,A -85,B 0,C 180,E1 -17408.786,E2 -17408.786} C_VEL
LIN {X 0,Y 279.43,Z 382.103,A -85,B 0,C 180,E1 -17412.051,E2 -17412.051} C_VEL
LIN {X 0,Y 278.084,Z 375.072,A -85,B 0,C 180,E1 -17415.972,E2 -17415.972} C_VEL
LIN {X 0,Y 277.253,Z 370.951,A -85,B 0,C 180,E1 -17418.53,E2 -17418.53} C_VEL
LIN {X 0,Y 277.272,Z 370.949,A -85,B 0,C 180,E1 -17422.532,E2 -17422.532} C_VEL
LIN {X 0,Y 277.251,Z 370.95,A -85,B 0,C 180,E1 -17426.105,E2 -17426.105} C_VEL
LIN {X 0,Y 277.266,Z 370.946,A -85,B 0,C 180,E1 -17429.539,E2 -17429.539} C_VEL
LIN {X 0,Y 277.361,Z 370.938,A -85,B 0,C 180,E1 -17432.864,E2 -17432.864} C_VEL
LIN {X 0,Y 277.333,Z 370.939,A -85,B 0,C 180,E1 -17436.08,E2 -17436.08} C_VEL
LIN {X 0,Y 277.35,Z 370.94,A -85,B 0,C 180,E1 -17440.767,E2 -17440.767} C_VEL
LIN {X 0,Y 277.44,Z 370.925,A -85,B 0,C 180,E1 -17445.326,E2 -17445.326} C_VEL
LIN {X 0,Y 277.512,Z 370.916,A -85,B 0,C 180,E1 -17449.789,E2 -17449.789} C_VEL
LIN {X 0,Y 277.66,Z 370.898,A -85,B 0,C 180,E1 -17452.73,E2 -17452.73} C_VEL
LIN {X 0,Y 277.827,Z 370.873,A -85,B 0,C 180,E1 -17458.551,E2 -17458.551} C_VEL
LIN {X 0,Y 277.827,Z 370.875,A -85,B 0,C 180,E1 -17461.45,E2 -17461.45} C_VEL
LIN {X 0,Y 277.66,Z 370.89,A -85,B 0,C 180,E1 -17467.271,E2 -17467.271} C_VEL
LIN {X 0,Y 277.513,Z 370.917,A -85,B 0,C 180,E1 -17470.211,E2 -17470.211} C_VEL
LIN {X 0,Y 277.441,Z 370.918,A -85,B 0,C 180,E1 -17474.674,E2 -17474.674} C_VEL
LIN {X 0,Y 277.351,Z 370.935,A -85,B 0,C 180,E1 -17479.234,E2 -17479.234} C_VEL
LIN {X 0,Y 277.335,Z 370.937,A -85,B 0,C 180,E1 -17483.92,E2 -17483.92} C_VEL
LIN {X 0,Y 277.331,Z 370.941,A -85,B 0,C 180,E1 -17487.505,E2 -17487.505} C_VEL
LIN {X 0,Y 277.278,Z 370.94,A -85,B 0,C 180,E1 -17490.481,E2 -17490.481} C_VEL
LIN {X 0,Y 277.26,Z 370.948,A -85,B 0,C 180,E1 -17493.894,E2 -17493.894} C_VEL
LIN {X 0,Y 277.288,Z 370.947,A -85,B 0,C 180,E1 -17497.467,E2 -17497.467} C_VEL
LIN {X 0,Y 277.216,Z 370.954,A -85,B 0,C 180,E1 -17501.236,E2 -17501.236} C_VEL
LIN {X 0,Y 277.223,Z 370.953,A -85,B 0,C 180,E1 -17505.223,E2 -17505.223} C_VEL
LIN {X 0,Y 277.229,Z 370.951,A -85,B 0,C 180,E1 -17509.512,E2 -17509.512} C_VEL
LIN {X 0,Y 277.274,Z 370.943,A -85,B 0,C 180,E1 -17512.53,E2 -17512.53} C_VEL
LIN {X 0,Y 277.253,Z 370.947,A -85,B 0,C 180,E1 -17516.104,E2 -17516.104} C_VEL
LIN {X 0,Y 277.267,Z 370.947,A -85,B 0,C 180,E1 -17519.538,E2 -17519.538} C_VEL
LIN {X 0,Y 277.365,Z 370.937,A -85,B 0,C 180,E1 -17522.864,E2 -17522.864} C_VEL
LIN {X 0,Y 277.335,Z 370.937,A -85,B 0,C 180,E1 -17526.079,E2 -17526.079} C_VEL
LIN {X 0,Y 277.351,Z 370.937,A -85,B 0,C 180,E1 -17530.766,E2 -17530.766} C_VEL
LIN {X 0,Y 277.451,Z 370.943,A -85,B 0,C 180,E1 -17534.275,E2 -17534.275} C_VEL
LIN {X 0,Y 281.676,Z 383.209,A -85,B 0,C 180,E1 -17535.551,E2 -17535.551} C_VEL
LIN {X 0,Y 284.528,Z 392.757,A -85,B 0,C 180,E1 -17536.726,E2 -17536.726} C_VEL
LIN {X 0,Y 285.43,Z 396.233,A -85,B 0,C 180,E1 -17537.196,E2 -17537.196} C_VEL
LIN {X 0,Y 284.713,Z 404.784,A -85,B 0,C 180,E1 -17538.249,E2 -17538.249} C_VEL
LIN {X 0,Y 283.444,Z 415.283,A -85,B 0,C 180,E1 -17539.823,E2 -17539.823} C_VEL
LIN {X 0,Y 282.081,Z 425.605,A -85,B 0,C 180,E1 -17541.762,E2 -17541.762} C_VEL
LIN {X 0,Y 280.637,Z 434.567,A -85,B 0,C 180,E1 -17543.889,E2 -17543.889} C_VEL
LIN {X 0,Y 279.463,Z 441.791,A -85,B 0,C 180,E1 -17546.033,E2 -17546.033} C_VEL
LIN {X 0,Y 278.43,Z 448.424,A -85,B 0,C 180,E1 -17548.553,E2 -17548.553} C_VEL
LIN {X 0,Y 277.789,Z 452.811,A -85,B 0,C 180,E1 -17550.724,E2 -17550.724} C_VEL
LIN {X 0,Y 277.212,Z 456.172,A -85,B 0,C 180,E1 -17552.905,E2 -17552.905} C_VEL
LIN {X 0,Y 277.103,Z 459.091,A -85,B 0,C 180,E1 -17555.822,E2 -17555.822} C_VEL
LIN {X 0,Y 277.107,Z 460.404,A -85,B 0,C 180,E1 -17558.455,E2 -17558.455} C_VEL
LIN {X 0,Y 277.235,Z 460.54,A -85,B 0,C 180,E1 -17560.22,E2 -17560.22} C_VEL
LIN {X 0,Y 277.77,Z 459.565,A -85,B 0,C 180,E1 -17563.161,E2 -17563.161} C_VEL
LIN {X 0,Y 278.189,Z 458.443,A -85,B 0,C 180,E1 -17564.632,E2 -17564.632} C_VEL
LIN {X 0,Y 279.131,Z 455.885,A -85,B 0,C 180,E1 -17566.907,E2 -17566.907} C_VEL
LIN {X 0,Y 280.219,Z 452.523,A -85,B 0,C 180,E1 -17569.028,E2 -17569.028} C_VEL
LIN {X 0,Y 281.573,Z 447.928,A -85,B 0,C 180,E1 -17571.217,E2 -17571.217} C_VEL
LIN {X 0,Y 283.504,Z 440.946,A -85,B 0,C 180,E1 -17573.754,E2 -17573.754} C_VEL
LIN {X 0,Y 285.501,Z 433.278,A -85,B 0,C 180,E1 -17575.908,E2 -17575.908} C_VEL
LIN {X 0,Y 287.693,Z 423.653,A -85,B 0,C 180,E1 -17578.035,E2 -17578.035} C_VEL
LIN {X 0,Y 289.701,Z 413.45,A -85,B 0,C 180,E1 -17579.822,E2 -17579.822} C_VEL
LIN {X 0,Y 290.843,Z 407.042,A -85,B 0,C 180,E1 -17580.742,E2 -17580.742} C_VEL
LIN {X 0,Y 290.116,Z 403.488,A -85,B 0,C 180,E1 -17581.358,E2 -17581.358} C_VEL
LIN {X 0,Y 287.013,Z 393.992,A -85,B 0,C 180,E1 -17582.969,E2 -17582.969} C_VEL
LIN {X 0,Y 283.343,Z 384.453,A -85,B 0,C 180,E1 -17584.438,E2 -17584.438} C_VEL
LIN {X 0,Y 278.235,Z 373.684,A -85,B 0,C 180,E1 -17585.992,E2 -17585.992} C_VEL
LIN {X 0,Y 277.289,Z 370.947,A -85,B 0,C 180,E1 -17586.343,E2 -17586.343} C_VEL
LIN {X 0,Y 277.222,Z 370.953,A -85,B 0,C 180,E1 -17590.487,E2 -17590.487} C_VEL
LIN {X 0,Y 277.202,Z 370.955,A -85,B 0,C 180,E1 -17594.773,E2 -17594.773} C_VEL
LIN {X 0,Y 277.239,Z 370.955,A -85,B 0,C 180,E1 -17598.768,E2 -17598.768} C_VEL
LIN {X 0,Y 277.288,Z 370.947,A -85,B 0,C 180,E1 -17602.533,E2 -17602.533} C_VEL
LIN {X 0,Y 277.253,Z 370.951,A -85,B 0,C 180,E1 -17606.104,E2 -17606.104} C_VEL
LIN {X 0,Y 277.259,Z 370.908,A -85,B 0,C 180,E1 -17609.538,E2 -17609.538} C_VEL
LIN {X 0,Y 277.356,Z 370.927,A -85,B 0,C 180,E1 -17612.863,E2 -17612.863} C_VEL
LIN {X 0,Y 277.326,Z 370.931,A -85,B 0,C 180,E1 -17616.079,E2 -17616.079} C_VEL
LIN {X 0,Y 277.342,Z 370.935,A -85,B 0,C 180,E1 -17620.766,E2 -17620.766} C_VEL
LIN {X 0,Y 277.432,Z 370.929,A -85,B 0,C 180,E1 -17625.325,E2 -17625.325} C_VEL
LIN {X 0,Y 277.504,Z 370.915,A -85,B 0,C 180,E1 -17629.788,E2 -17629.788} C_VEL
LIN {X 0,Y 277.65,Z 370.896,A -85,B 0,C 180,E1 -17632.729,E2 -17632.729} C_VEL
LIN {X 0,Y 277.822,Z 370.875,A -85,B 0,C 180,E1 -17638.55,E2 -17638.55} C_VEL
LIN {X 0,Y 277.822,Z 370.875,A -85,B 0,C 180,E1 -17641.449,E2 -17641.449} C_VEL
LIN {X 0,Y 277.649,Z 370.901,A -85,B 0,C 180,E1 -17647.271,E2 -17647.271} C_VEL
LIN {X 0,Y 277.502,Z 370.909,A -85,B 0,C 180,E1 -17650.211,E2 -17650.211} C_VEL
LIN {X 0,Y 277.41,Z 370.924,A -85,B 0,C 180,E1 -17653.122,E2 -17653.122} C_VEL
LIN {X 0,Y 276.765,Z 371.009,A -85,B 0,C 180,E1 -17654.334,E2 -17654.334} C_VEL
LIN {X 0,Y 273.848,Z 371.373,A -85,B 0,C 180,E1 -17656.304,E2 -17656.304} C_VEL
LIN {X 0,Y 271.374,Z 371.676,A -85,B 0,C 180,E1 -17657.906,E2 -17657.906} C_VEL
LIN {X 0,Y 270.348,Z 371.811,A -85,B 0,C 180,E1 -17659.15,E2 -17659.15} C_VEL
LIN {X 0,Y 270.285,Z 371.816,A -85,B 0,C 180,E1 -17659.572,E2 -17659.572} C_VEL
LIN {X 0,Y 270.27,Z 371.821,A -85,B 0,C 180,E1 -17664.586,E2 -17664.586} C_VEL
LIN {X 0,Y 270.268,Z 371.825,A -85,B 0,C 180,E1 -17667.909,E2 -17667.909} C_VEL
LIN {X 0,Y 270.18,Z 371.834,A -85,B 0,C 180,E1 -17671.349,E2 -17671.349} C_VEL
LIN {X 0,Y 270.258,Z 372.007,A -85,B 0,C 180,E1 -17674.724,E2 -17674.724} C_VEL
LIN {X 0,Y 271.331,Z 376.904,A -85,B 0,C 180,E1 -17678.436,E2 -17678.436} C_VEL
LIN {X 0,Y 272.377,Z 382.251,A -85,B 0,C 180,E1 -17682.134,E2 -17682.134} C_VEL
LIN {X 0,Y 273.586,Z 388.415,A -85,B 0,C 180,E1 -17686.087,E2 -17686.087} C_VEL
LIN {X 0,Y 274.851,Z 395.477,A -85,B 0,C 180,E1 -17690.265,E2 -17690.265} C_VEL
LIN {X 0,Y 275.034,Z 397.211,A -85,B 0,C 180,E1 -17691.242,E2 -17691.242} C_VEL
LIN {X 0,Y 274.318,Z 400.914,A -85,B 0,C 180,E1 -17693.173,E2 -17693.173} C_VEL
LIN {X 0,Y 272.646,Z 408.922,A -85,B 0,C 180,E1 -17697.228,E2 -17697.228} C_VEL
LIN {X 0,Y 271.532,Z 415.205,A -85,B 0,C 180,E1 -17700.371,E2 -17700.371} C_VEL
LIN {X 0,Y 274.262,Z 427.51,A -85,B 0,C 180,E1 -17701.301,E2 -17701.301} C_VEL
LIN {X 0,Y 276.254,Z 438.613,A -85,B 0,C 180,E1 -17702.296,E2 -17702.296} C_VEL
LIN {X 0,Y 277.583,Z 450.911,A -85,B 0,C 180,E1 -17703.564,E2 -17703.564} C_VEL
LIN {X 0,Y 278.18,Z 462.992,A -85,B 0,C 180,E1 -17705.035,E2 -17705.035} C_VEL
LIN {X 0,Y 277.871,Z 473.471,A -85,B 0,C 180,E1 -17706.526,E2 -17706.526} C_VEL
LIN {X 0,Y 276.985,Z 482.514,A -85,B 0,C 180,E1 -17708.023,E2 -17708.023} C_VEL
LIN {X 0,Y 275.403,Z 490.09,A -85,B 0,C 180,E1 -17709.46,E2 -17709.46} C_VEL
LIN {X 0,Y 273.409,Z 498.084,A -85,B 0,C 180,E1 -17711.259,E2 -17711.259} C_VEL
LIN {X 0,Y 271.605,Z 505.974,A -85,B 0,C 180,E1 -17713.464,E2 -17713.464} C_VEL
LIN {X 0,Y 270.678,Z 510.375,A -85,B 0,C 180,E1 -17714.952,E2 -17714.952} C_VEL
LIN {X 0,Y 269.59,Z 515.914,A -85,B 0,C 180,E1 -17717.199,E2 -17717.199} C_VEL
LIN {X 0,Y 268.95,Z 520.3,A -85,B 0,C 180,E1 -17719.461,E2 -17719.461} C_VEL
LIN {X 0,Y 268.813,Z 522.669,A -85,B 0,C 180,E1 -17720.976,E2 -17720.976} C_VEL
LIN {X 0,Y 268.858,Z 525.499,A -85,B 0,C 180,E1 -17723.377,E2 -17723.377} C_VEL
LIN {X 0,Y 269.105,Z 527.112,A -85,B 0,C 180,E1 -17725.507,E2 -17725.507} C_VEL
LIN {X 0,Y 269.395,Z 527.796,A -85,B 0,C 180,E1 -17727.01,E2 -17727.01} C_VEL
LIN {X 0,Y 269.436,Z 528.007,A -85,B 0,C 180,E1 -17728.506,E2 -17728.506} C_VEL
LIN {X 0,Y 269.556,Z 527.805,A -85,B 0,C 180,E1 -17730.001,E2 -17730.001} C_VEL
LIN {X 0,Y 269.497,Z 527.175,A -85,B 0,C 180,E1 -17731.495,E2 -17731.495} C_VEL
LIN {X 0,Y 269.5,Z 526.142,A -85,B 0,C 180,E1 -17732.991,E2 -17732.991} C_VEL
LIN {X 0,Y 269.307,Z 524.619,A -85,B 0,C 180,E1 -17734.491,E2 -17734.491} C_VEL
LIN {X 0,Y 269.037,Z 521.157,A -85,B 0,C 180,E1 -17736.944,E2 -17736.944} C_VEL
LIN {X 0,Y 268.997,Z 515.573,A -85,B 0,C 180,E1 -17739.779,E2 -17739.779} C_VEL
LIN {X 0,Y 269.545,Z 508.617,A -85,B 0,C 180,E1 -17742.423,E2 -17742.423} C_VEL
LIN {X 0,Y 270.342,Z 501.041,A -85,B 0,C 180,E1 -17744.684,E2 -17744.684} C_VEL
LIN {X 0,Y 271.371,Z 493.353,A -85,B 0,C 180,E1 -17746.553,E2 -17746.553} C_VEL
LIN {X 0,Y 272.534,Z 486.077,A -85,B 0,C 180,E1 -17748.027,E2 -17748.027} C_VEL
LIN {X 0,Y 273.521,Z 477.402,A -85,B 0,C 180,E1 -17749.515,E2 -17749.515} C_VEL
LIN {X 0,Y 273.587,Z 466.618,A -85,B 0,C 180,E1 -17751.079,E2 -17751.079} C_VEL
LIN {X 0,Y 273.432,Z 454.57,A -85,B 0,C 180,E1 -17752.496,E2 -17752.496} C_VEL
LIN {X 0,Y 272.829,Z 442.246,A -85,B 0,C 180,E1 -17753.638,E2 -17753.638} C_VEL
LIN {X 0,Y 271.604,Z 429.571,A -85,B 0,C 180,E1 -17754.554,E2 -17754.554} C_VEL
LIN {X 0,Y 269.865,Z 417.312,A -85,B 0,C 180,E1 -17755.228,E2 -17755.228} C_VEL
LIN {X 0,Y 270.913,Z 408.291,A -85,B 0,C 180,E1 -17759.532,E2 -17759.532} C_VEL
LIN {X 0,Y 272.118,Z 399.86,A -85,B 0,C 180,E1 -17763.61,E2 -17763.61} C_VEL
LIN {X 0,Y 273.35,Z 392.624,A -85,B 0,C 180,E1 -17767.153,E2 -17767.153} C_VEL
LIN {X 0,Y 273.5,Z 389.408,A -85,B 0,C 180,E1 -17768.773,E2 -17768.773} C_VEL
LIN {X 0,Y 272.453,Z 383.304,A -85,B 0,C 180,E1 -17772.121,E2 -17772.121} C_VEL
LIN {X 0,Y 270.967,Z 375.59,A -85,B 0,C 180,E1 -17776.573,E2 -17776.573} C_VEL
LIN {X 0,Y 270.213,Z 371.828,A -85,B 0,C 180,E1 -17778.963,E2 -17778.963} C_VEL
LIN {X 0,Y 270.222,Z 371.829,A -85,B 0,C 180,E1 -17783.26,E2 -17783.26} C_VEL
LIN {X 0,Y 270.207,Z 371.83,A -85,B 0,C 180,E1 -17786.893,E2 -17786.893} C_VEL
LIN {X 0,Y 270.2,Z 371.828,A -85,B 0,C 180,E1 -17790.383,E2 -17790.383} C_VEL
LIN {X 0,Y 270.266,Z 371.819,A -85,B 0,C 180,E1 -17793.764,E2 -17793.764} C_VEL
LIN {X 0,Y 270.238,Z 371.825,A -85,B 0,C 180,E1 -17797.039,E2 -17797.039} C_VEL
LIN {X 0,Y 270.307,Z 371.816,A -85,B 0,C 180,E1 -17800.245,E2 -17800.245} C_VEL
LIN {X 0,Y 270.408,Z 371.802,A -85,B 0,C 180,E1 -17804.936,E2 -17804.936} C_VEL
LIN {X 0,Y 270.447,Z 371.795,A -85,B 0,C 180,E1 -17809.519,E2 -17809.519} C_VEL
LIN {X 0,Y 270.618,Z 371.777,A -85,B 0,C 180,E1 -17812.539,E2 -17812.539} C_VEL
LIN {X 0,Y 270.793,Z 371.748,A -85,B 0,C 180,E1 -17818.513,E2 -17818.513} C_VEL
LIN {X 0,Y 270.793,Z 371.751,A -85,B 0,C 180,E1 -17821.488,E2 -17821.488} C_VEL
LIN {X 0,Y 270.618,Z 371.767,A -85,B 0,C 180,E1 -17827.461,E2 -17827.461} C_VEL
LIN {X 0,Y 270.448,Z 371.796,A -85,B 0,C 180,E1 -17830.481,E2 -17830.481} C_VEL
LIN {X 0,Y 270.409,Z 371.793,A -85,B 0,C 180,E1 -17835.065,E2 -17835.065} C_VEL
LIN {X 0,Y 270.308,Z 371.816,A -85,B 0,C 180,E1 -17839.755,E2 -17839.755} C_VEL
LIN {X 0,Y 270.28,Z 371.814,A -85,B 0,C 180,E1 -17844.585,E2 -17844.585} C_VEL
LIN {X 0,Y 270.276,Z 371.817,A -85,B 0,C 180,E1 -17847.909,E2 -17847.909} C_VEL
LIN {X 0,Y 270.191,Z 371.825,A -85,B 0,C 180,E1 -17851.348,E2 -17851.348} C_VEL
LIN {X 0,Y 270.221,Z 371.823,A -85,B 0,C 180,E1 -17854.903,E2 -17854.903} C_VEL
LIN {X 0,Y 270.228,Z 371.821,A -85,B 0,C 180,E1 -17858.717,E2 -17858.717} C_VEL
LIN {X 0,Y 270.178,Z 371.831,A -85,B 0,C 180,E1 -17863.25,E2 -17863.25} C_VEL
LIN {X 0,Y 270.18,Z 371.83,A -85,B 0,C 180,E1 -17867.442,E2 -17867.442} C_VEL
LIN {X 0,Y 270.213,Z 371.826,A -85,B 0,C 180,E1 -17871.374,E2 -17871.374} C_VEL
LIN {X 0,Y 270.208,Z 371.827,A -85,B 0,C 180,E1 -17875.094,E2 -17875.094} C_VEL
LIN {X 0,Y 270.206,Z 371.828,A -85,B 0,C 180,E1 -17879.13,E2 -17879.13} C_VEL
LIN {X 0,Y 270.271,Z 371.818,A -85,B 0,C 180,E1 -17882.145,E2 -17882.145} C_VEL
LIN {X 0,Y 270.283,Z 371.816,A -85,B 0,C 180,E1 -17885.518,E2 -17885.518} C_VEL
LIN {X 0,Y 270.308,Z 371.814,A -85,B 0,C 180,E1 -17890.244,E2 -17890.244} C_VEL
LIN {X 0,Y 270.364,Z 371.868,A -85,B 0,C 180,E1 -17893.71,E2 -17893.71} C_VEL
LIN {X 0,Y 274.566,Z 383.548,A -85,B 0,C 180,E1 -17894.979,E2 -17894.979} C_VEL
LIN {X 0,Y 277.878,Z 394.756,A -85,B 0,C 180,E1 -17896.402,E2 -17896.402} C_VEL
LIN {X 0,Y 278.739,Z 398.123,A -85,B 0,C 180,E1 -17896.883,E2 -17896.883} C_VEL
LIN {X 0,Y 277.552,Z 409.053,A -85,B 0,C 180,E1 -17898.312,E2 -17898.312} C_VEL
LIN {X 0,Y 276.43,Z 417.913,A -85,B 0,C 180,E1 -17899.747,E2 -17899.747} C_VEL
LIN {X 0,Y 275.142,Z 427.026,A -85,B 0,C 180,E1 -17901.553,E2 -17901.553} C_VEL
LIN {X 0,Y 273.683,Z 435.886,A -85,B 0,C 180,E1 -17903.733,E2 -17903.733} C_VEL
LIN {X 0,Y 272.443,Z 443.037,A -85,B 0,C 180,E1 -17905.931,E2 -17905.931} C_VEL
LIN {X 0,Y 271.68,Z 447.864,A -85,B 0,C 180,E1 -17907.775,E2 -17907.775} C_VEL
LIN {X 0,Y 270.922,Z 452.571,A -85,B 0,C 180,E1 -17909.999,E2 -17909.999} C_VEL
LIN {X 0,Y 270.319,Z 456.202,A -85,B 0,C 180,E1 -17912.234,E2 -17912.234} C_VEL
LIN {X 0,Y 270.06,Z 458.824,A -85,B 0,C 180,E1 -17914.477,E2 -17914.477} C_VEL
LIN {X 0,Y 270.052,Z 460.062,A -85,B 0,C 180,E1 -17915.974,E2 -17915.974} C_VEL
LIN {X 0,Y 270.068,Z 461.278,A -85,B 0,C 180,E1 -17918.549,E2 -17918.549} C_VEL
LIN {X 0,Y 270.228,Z 461.405,A -85,B 0,C 180,E1 -17920.488,E2 -17920.488} C_VEL
LIN {X 0,Y 270.473,Z 461.083,A -85,B 0,C 180,E1 -17921.997,E2 -17921.997} C_VEL
LIN {X 0,Y 270.839,Z 460.357,A -85,B 0,C 180,E1 -17923.504,E2 -17923.504} C_VEL
LIN {X 0,Y 271.281,Z 459.199,A -85,B 0,C 180,E1 -17925.014,E2 -17925.014} C_VEL
LIN {X 0,Y 272.239,Z 456.758,A -85,B 0,C 180,E1 -17927.218,E2 -17927.218} C_VEL
LIN {X 0,Y 273.45,Z 453.164,A -85,B 0,C 180,E1 -17929.518,E2 -17929.518} C_VEL
LIN {X 0,Y 274.885,Z 448.504,A -85,B 0,C 180,E1 -17931.759,E2 -17931.759} C_VEL
LIN {X 0,Y 276.62,Z 442.557,A -85,B 0,C 180,E1 -17933.984,E2 -17933.984} C_VEL
LIN {X 0,Y 278.711,Z 435.092,A -85,B 0,C 180,E1 -17936.184,E2 -17936.184} C_VEL
LIN {X 0,Y 280.592,Z 427.409,A -85,B 0,C 180,E1 -17938.009,E2 -17938.009} C_VEL
LIN {X 0,Y 282.588,Z 417.945,A -85,B 0,C 180,E1 -17939.827,E2 -17939.827} C_VEL
LIN {X 0,Y 284.381,Z 408.653,A -85,B 0,C 180,E1 -17941.263,E2 -17941.263} C_VEL
LIN {X 0,Y 281.865,Z 399.838,A -85,B 0,C 180,E1 -17942.879,E2 -17942.879} C_VEL
LIN {X 0,Y 277.835,Z 388.669,A -85,B 0,C 180,E1 -17944.743,E2 -17944.743} C_VEL
LIN {X 0,Y 272.924,Z 377.909,A -85,B 0,C 180,E1 -17946.417,E2 -17946.417} C_VEL
LIN {X 0,Y 270.403,Z 372.752,A -85,B 0,C 180,E1 -17947.157,E2 -17947.157} C_VEL
LIN {X 0,Y 270.245,Z 371.825,A -85,B 0,C 180,E1 -17947.298,E2 -17947.298} C_VEL
LIN {X 0,Y 270.168,Z 371.834,A -85,B 0,C 180,E1 -17951.027,E2 -17951.027} C_VEL
LIN {X 0,Y 270.157,Z 371.836,A -85,B 0,C 180,E1 -17955.38,E2 -17955.38} C_VEL
LIN {X 0,Y 270.235,Z 371.824,A -85,B 0,C 180,E1 -17959.444,E2 -17959.444} C_VEL
LIN {X 0,Y 270.256,Z 371.816,A -85,B 0,C 180,E1 -17963.72,E2 -17963.72} C_VEL
LIN {X 0,Y 270.203,Z 371.822,A -85,B 0,C 180,E1 -17966.892,E2 -17966.892} C_VEL
LIN {X 0,Y 270.194,Z 371.787,A -85,B 0,C 180,E1 -17970.382,E2 -17970.382} C_VEL
LIN {X 0,Y 270.261,Z 371.818,A -85,B 0,C 180,E1 -17973.763,E2 -17973.763} C_VEL
LIN {X 0,Y 270.23,Z 371.811,A -85,B 0,C 180,E1 -17977.038,E2 -17977.038} C_VEL
LIN {X 0,Y 270.299,Z 371.815,A -85,B 0,C 180,E1 -17980.244,E2 -17980.244} C_VEL
LIN {X 0,Y 270.4,Z 371.804,A -85,B 0,C 180,E1 -17984.935,E2 -17984.935} C_VEL
LIN {X 0,Y 270.439,Z 371.795,A -85,B 0,C 180,E1 -17989.518,E2 -17989.518} C_VEL
LIN {X 0,Y 270.608,Z 371.774,A -85,B 0,C 180,E1 -17992.538,E2 -17992.538} C_VEL
LIN {X 0,Y 270.788,Z 371.751,A -85,B 0,C 180,E1 -17998.512,E2 -17998.512} C_VEL
LIN {X 0,Y 270.787,Z 371.751,A -85,B 0,C 180,E1 -18001.487,E2 -18001.487} C_VEL
LIN {X 0,Y 270.607,Z 371.779,A -85,B 0,C 180,E1 -18007.461,E2 -18007.461} C_VEL
LIN {X 0,Y 270.437,Z 371.79,A -85,B 0,C 180,E1 -18010.481,E2 -18010.481} C_VEL
LIN {X 0,Y 270.399,Z 371.801,A -85,B 0,C 180,E1 -18015.065,E2 -18015.065} C_VEL
LIN {X 0,Y 270.285,Z 371.816,A -85,B 0,C 180,E1 -18019.572,E2 -18019.572} C_VEL
LIN {X 0,Y 269.664,Z 371.902,A -85,B 0,C 180,E1 -18020.815,E2 -18020.815} C_VEL
LIN {X 0,Y 266.79,Z 372.262,A -85,B 0,C 180,E1 -18022.84,E2 -18022.84} C_VEL
LIN {X 0,Y 264.316,Z 372.565,A -85,B 0,C 180,E1 -18024.487,E2 -18024.487} C_VEL
LIN {X 0,Y 263.253,Z 372.697,A -85,B 0,C 180,E1 -18025.765,E2 -18025.765} C_VEL
LIN {X 0,Y 263.167,Z 372.705,A -85,B 0,C 180,E1 -18026.198,E2 -18026.198} C_VEL
LIN {X 0,Y 263.176,Z 372.707,A -85,B 0,C 180,E1 -18028.73,E2 -18028.73} C_VEL
LIN {X 0,Y 263.164,Z 372.705,A -85,B 0,C 180,E1 -18033.193,E2 -18033.193} C_VEL
LIN {X 0,Y 263.198,Z 372.89,A -85,B 0,C 180,E1 -18033.818,E2 -18033.818} C_VEL
LIN {X 0,Y 264.279,Z 377.829,A -85,B 0,C 180,E1 -18037.708,E2 -18037.708} C_VEL
LIN {X 0,Y 265.319,Z 383.048,A -85,B 0,C 180,E1 -18041.469,E2 -18041.469} C_VEL
LIN {X 0,Y 266.684,Z 390.018,A -85,B 0,C 180,E1 -18046.092,E2 -18046.092} C_VEL
LIN {X 0,Y 267.89,Z 396.934,A -85,B 0,C 180,E1 -18050.298,E2 -18050.298} C_VEL
LIN {X 0,Y 267.863,Z 399.821,A -85,B 0,C 180,E1 -18051.917,E2 -18051.917} C_VEL
LIN {X 0,Y 265.96,Z 408.179,A -85,B 0,C 180,E1 -18056.296,E2 -18056.296} C_VEL
LIN {X 0,Y 264.782,Z 414.222,A -85,B 0,C 180,E1 -18059.414,E2 -18059.414} C_VEL
LIN {X 0,Y 266.436,Z 421.396,A -85,B 0,C 180,E1 -18059.964,E2 -18059.964} C_VEL
LIN {X 0,Y 269.111,Z 434.598,A -85,B 0,C 180,E1 -18061.138,E2 -18061.138} C_VEL
LIN {X 0,Y 270.746,Z 447.521,A -85,B 0,C 180,E1 -18062.481,E2 -18062.481} C_VEL
LIN {X 0,Y 271.45,Z 459.095,A -85,B 0,C 180,E1 -18063.888,E2 -18063.888} C_VEL
LIN {X 0,Y 271.417,Z 469.243,A -85,B 0,C 180,E1 -18065.315,E2 -18065.315} C_VEL
LIN {X 0,Y 270.562,Z 479.963,A -85,B 0,C 180,E1 -18067.069,E2 -18067.069} C_VEL
LIN {X 0,Y 269.201,Z 487.813,A -85,B 0,C 180,E1 -18068.563,E2 -18068.563} C_VEL
LIN {X 0,Y 266.636,Z 497.53,A -85,B 0,C 180,E1 -18070.764,E2 -18070.764} C_VEL
LIN {X 0,Y 264.726,Z 505.336,A -85,B 0,C 180,E1 -18073.022,E2 -18073.022} C_VEL
LIN {X 0,Y 263.813,Z 509.718,A -85,B 0,C 180,E1 -18074.551,E2 -18074.551} C_VEL
LIN {X 0,Y 262.62,Z 515.207,A -85,B 0,C 180,E1 -18076.853,E2 -18076.853} C_VEL
LIN {X 0,Y 261.918,Z 519.55,A -85,B 0,C 180,E1 -18079.175,E2 -18079.175} C_VEL
LIN {X 0,Y 261.744,Z 521.893,A -85,B 0,C 180,E1 -18080.73,E2 -18080.73} C_VEL
LIN {X 0,Y 261.863,Z 525.22,A -85,B 0,C 180,E1 -18083.838,E2 -18083.838} C_VEL
LIN {X 0,Y 262.322,Z 526.939,A -85,B 0,C 180,E1 -18086.93,E2 -18086.93} C_VEL
LIN {X 0,Y 262.39,Z 527.125,A -85,B 0,C 180,E1 -18088.466,E2 -18088.466} C_VEL
LIN {X 0,Y 262.51,Z 526.906,A -85,B 0,C 180,E1 -18090.001,E2 -18090.001} C_VEL
LIN {X 0,Y 262.448,Z 526.258,A -85,B 0,C 180,E1 -18091.536,E2 -18091.536} C_VEL
LIN {X 0,Y 262.45,Z 525.204,A -85,B 0,C 180,E1 -18093.071,E2 -18093.071} C_VEL
LIN {X 0,Y 262.097,Z 522.705,A -85,B 0,C 180,E1 -18095.386,E2 -18095.386} C_VEL
LIN {X 0,Y 261.915,Z 519.167,A -85,B 0,C 180,E1 -18097.712,E2 -18097.712} C_VEL
LIN {X 0,Y 261.958,Z 514.51,A -85,B 0,C 180,E1 -18100.044,E2 -18100.044} C_VEL
LIN {X 0,Y 262.56,Z 507.483,A -85,B 0,C 180,E1 -18102.759,E2 -18102.759} C_VEL
LIN {X 0,Y 263.419,Z 499.854,A -85,B 0,C 180,E1 -18105.079,E2 -18105.079} C_VEL
LIN {X 0,Y 264.557,Z 492.112,A -85,B 0,C 180,E1 -18106.992,E2 -18106.992} C_VEL
LIN {X 0,Y 265.99,Z 482.749,A -85,B 0,C 180,E1 -18108.886,E2 -18108.886} C_VEL
LIN {X 0,Y 266.565,Z 475.943,A -85,B 0,C 180,E1 -18110.045,E2 -18110.045} C_VEL
LIN {X 0,Y 266.633,Z 465.019,A -85,B 0,C 180,E1 -18111.656,E2 -18111.656} C_VEL
LIN {X 0,Y 266.546,Z 453.12,A -85,B 0,C 180,E1 -18113.071,E2 -18113.071} C_VEL
LIN {X 0,Y 265.871,Z 439.941,A -85,B 0,C 180,E1 -18114.302,E2 -18114.302} C_VEL
LIN {X 0,Y 264.381,Z 426.439,A -85,B 0,C 180,E1 -18115.286,E2 -18115.286} C_VEL
LIN {X 0,Y 262.894,Z 416.45,A -85,B 0,C 180,E1 -18115.836,E2 -18115.836} C_VEL
LIN {X 0,Y 264.049,Z 407.227,A -85,B 0,C 180,E1 -18120.38,E2 -18120.38} C_VEL
LIN {X 0,Y 265.484,Z 398.236,A -85,B 0,C 180,E1 -18124.851,E2 -18124.851} C_VEL
LIN {X 0,Y 266.415,Z 392.67,A -85,B 0,C 180,E1 -18127.684,E2 -18127.684} C_VEL
LIN {X 0,Y 266.376,Z 389.663,A -85,B 0,C 180,E1 -18129.289,E2 -18129.289} C_VEL
LIN {X 0,Y 265.192,Z 383.143,A -85,B 0,C 180,E1 -18132.973,E2 -18132.973} C_VEL
LIN {X 0,Y 263.848,Z 376.121,A -85,B 0,C 180,E1 -18137.217,E2 -18137.217} C_VEL
LIN {X 0,Y 263.16,Z 372.706,A -85,B 0,C 180,E1 -18139.436,E2 -18139.436} C_VEL
LIN {X 0,Y 263.187,Z 372.706,A -85,B 0,C 180,E1 -18143.237,E2 -18143.237} C_VEL
LIN {X 0,Y 263.137,Z 372.707,A -85,B 0,C 180,E1 -18147.713,E2 -18147.713} C_VEL
LIN {X 0,Y 263.2,Z 372.698,A -85,B 0,C 180,E1 -18151.786,E2 -18151.786} C_VEL
LIN {X 0,Y 263.231,Z 372.697,A -85,B 0,C 180,E1 -18155.201,E2 -18155.201} C_VEL
LIN {X 0,Y 263.269,Z 372.691,A -85,B 0,C 180,E1 -18159.694,E2 -18159.694} C_VEL
LIN {X 0,Y 263.356,Z 372.683,A -85,B 0,C 180,E1 -18164.523,E2 -18164.523} C_VEL
LIN {X 0,Y 263.38,Z 372.676,A -85,B 0,C 180,E1 -18169.235,E2 -18169.235} C_VEL
LIN {X 0,Y 263.579,Z 372.654,A -85,B 0,C 180,E1 -18172.339,E2 -18172.339} C_VEL
LIN {X 0,Y 263.757,Z 372.624,A -85,B 0,C 180,E1 -18178.473,E2 -18178.473} C_VEL
LIN {X 0,Y 263.757,Z 372.627,A -85,B 0,C 180,E1 -18181.527,E2 -18181.527} C_VEL
LIN {X 0,Y 263.579,Z 372.644,A -85,B 0,C 180,E1 -18187.662,E2 -18187.662} C_VEL
LIN {X 0,Y 263.38,Z 372.675,A -85,B 0,C 180,E1 -18190.766,E2 -18190.766} C_VEL
LIN {X 0,Y 263.357,Z 372.672,A -85,B 0,C 180,E1 -18195.478,E2 -18195.478} C_VEL
LIN {X 0,Y 263.271,Z 372.689,A -85,B 0,C 180,E1 -18200.307,E2 -18200.307} C_VEL
LIN {X 0,Y 263.214,Z 372.695,A -85,B 0,C 180,E1 -18205.291,E2 -18205.291} C_VEL
LIN {X 0,Y 263.182,Z 372.698,A -85,B 0,C 180,E1 -18208.73,E2 -18208.73} C_VEL
LIN {X 0,Y 263.14,Z 372.705,A -85,B 0,C 180,E1 -18212.288,E2 -18212.288} C_VEL
LIN {X 0,Y 263.194,Z 372.699,A -85,B 0,C 180,E1 -18215.978,E2 -18215.978} C_VEL
LIN {X 0,Y 263.121,Z 372.708,A -85,B 0,C 180,E1 -18219.87,E2 -18219.87} C_VEL
LIN {X 0,Y 263.134,Z 372.705,A -85,B 0,C 180,E1 -18223.983,E2 -18223.983} C_VEL
LIN {X 0,Y 263.131,Z 372.705,A -85,B 0,C 180,E1 -18228.406,E2 -18228.406} C_VEL
LIN {X 0,Y 263.189,Z 372.702,A -85,B 0,C 180,E1 -18233.236,E2 -18233.236} C_VEL
LIN {X 0,Y 263.139,Z 372.706,A -85,B 0,C 180,E1 -18237.711,E2 -18237.711} C_VEL
LIN {X 0,Y 263.207,Z 372.698,A -85,B 0,C 180,E1 -18241.782,E2 -18241.782} C_VEL
LIN {X 0,Y 263.232,Z 372.697,A -85,B 0,C 180,E1 -18245.199,E2 -18245.199} C_VEL
LIN {X 0,Y 263.269,Z 372.69,A -85,B 0,C 180,E1 -18249.693,E2 -18249.693} C_VEL
LIN {X 0,Y 263.293,Z 372.69,A -85,B 0,C 180,E1 -18253.097,E2 -18253.097} C_VEL
LIN {X 0,Y 268.004,Z 385.726,A -85,B 0,C 180,E1 -18254.591,E2 -18254.591} C_VEL
LIN {X 0,Y 271.268,Z 396.905,A -85,B 0,C 180,E1 -18256.094,E2 -18256.094} C_VEL
LIN {X 0,Y 272.022,Z 400.014,A -85,B 0,C 180,E1 -18256.553,E2 -18256.553} C_VEL
LIN {X 0,Y 270.697,Z 410.736,A -85,B 0,C 180,E1 -18258.011,E2 -18258.011} C_VEL
LIN {X 0,Y 269.279,Z 421.37,A -85,B 0,C 180,E1 -18259.852,E2 -18259.852} C_VEL
LIN {X 0,Y 267.955,Z 430.031,A -85,B 0,C 180,E1 -18261.705,E2 -18261.705} C_VEL
LIN {X 0,Y 266.477,Z 438.504,A -85,B 0,C 180,E1 -18263.943,E2 -18263.943} C_VEL
LIN {X 0,Y 265.266,Z 445.278,A -85,B 0,C 180,E1 -18266.201,E2 -18266.201} C_VEL
LIN {X 0,Y 264.364,Z 450.701,A -85,B 0,C 180,E1 -18268.476,E2 -18268.476} C_VEL
LIN {X 0,Y 263.662,Z 454.973,A -85,B 0,C 180,E1 -18270.763,E2 -18270.763} C_VEL
LIN {X 0,Y 263.097,Z 458.217,A -85,B 0,C 180,E1 -18273.061,E2 -18273.061} C_VEL
LIN {X 0,Y 263.004,Z 461.031,A -85,B 0,C 180,E1 -18276.135,E2 -18276.135} C_VEL
LIN {X 0,Y 263.03,Z 462.152,A -85,B 0,C 180,E1 -18278.648,E2 -18278.648} C_VEL
LIN {X 0,Y 263.244,Z 462.268,A -85,B 0,C 180,E1 -18280.77,E2 -18280.77} C_VEL
LIN {X 0,Y 263.516,Z 461.92,A -85,B 0,C 180,E1 -18282.318,E2 -18282.318} C_VEL
LIN {X 0,Y 263.897,Z 461.143,A -85,B 0,C 180,E1 -18283.867,E2 -18283.867} C_VEL
LIN {X 0,Y 264.389,Z 459.957,A -85,B 0,C 180,E1 -18285.415,E2 -18285.415} C_VEL
LIN {X 0,Y 265.369,Z 457.62,A -85,B 0,C 180,E1 -18287.554,E2 -18287.554} C_VEL
LIN {X 0,Y 266.717,Z 453.805,A -85,B 0,C 180,E1 -18290.031,E2 -18290.031} C_VEL
LIN {X 0,Y 268.237,Z 449.081,A -85,B 0,C 180,E1 -18292.327,E2 -18292.327} C_VEL
LIN {X 0,Y 270.085,Z 443.062,A -85,B 0,C 180,E1 -18294.603,E2 -18294.603} C_VEL
LIN {X 0,Y 272.28,Z 435.507,A -85,B 0,C 180,E1 -18296.852,E2 -18296.852} C_VEL
LIN {X 0,Y 274.275,Z 427.701,A -85,B 0,C 180,E1 -18298.713,E2 -18298.713} C_VEL
LIN {X 0,Y 276.355,Z 418.101,A -85,B 0,C 180,E1 -18300.571,E2 -18300.571} C_VEL
LIN {X 0,Y 277.815,Z 411.244,A -85,B 0,C 180,E1 -18301.662,E2 -18301.662} C_VEL
LIN {X 0,Y 277.419,Z 408.655,A -85,B 0,C 180,E1 -18302.14,E2 -18302.14} C_VEL
LIN {X 0,Y 274.421,Z 398.871,A -85,B 0,C 180,E1 -18303.99,E2 -18303.99} C_VEL
LIN {X 0,Y 270.409,Z 388.371,A -85,B 0,C 180,E1 -18305.808,E2 -18305.808} C_VEL
LIN {X 0,Y 265.603,Z 378.25,A -85,B 0,C 180,E1 -18307.455,E2 -18307.455} C_VEL
LIN {X 0,Y 264.25,Z 375.67,A -85,B 0,C 180,E1 -18307.856,E2 -18307.856} C_VEL
LIN {X 0,Y 263.183,Z 372.702,A -85,B 0,C 180,E1 -18308.271,E2 -18308.271} C_VEL
LIN {X 0,Y 263.123,Z 372.707,A -85,B 0,C 180,E1 -18311.892,E2 -18311.892} C_VEL
LIN {X 0,Y 263.129,Z 372.711,A -85,B 0,C 180,E1 -18316.148,E2 -18316.148} C_VEL
LIN {X 0,Y 263.152,Z 372.703,A -85,B 0,C 180,E1 -18320.135,E2 -18320.135} C_VEL
LIN {X 0,Y 263.188,Z 372.696,A -85,B 0,C 180,E1 -18324.021,E2 -18324.021} C_VEL
LIN {X 0,Y 263.132,Z 372.69,A -85,B 0,C 180,E1 -18327.711,E2 -18327.711} C_VEL
LIN {X 0,Y 263.194,Z 372.674,A -85,B 0,C 180,E1 -18331.784,E2 -18331.784} C_VEL
LIN {X 0,Y 263.223,Z 372.694,A -85,B 0,C 180,E1 -18335.199,E2 -18335.199} C_VEL
LIN {X 0,Y 263.26,Z 372.692,A -85,B 0,C 180,E1 -18339.693,E2 -18339.693} C_VEL
LIN {X 0,Y 263.348,Z 372.682,A -85,B 0,C 180,E1 -18344.521,E2 -18344.521} C_VEL
LIN {X 0,Y 263.371,Z 372.677,A -85,B 0,C 180,E1 -18349.234,E2 -18349.234} C_VEL
LIN {X 0,Y 263.569,Z 372.652,A -85,B 0,C 180,E1 -18352.338,E2 -18352.338} C_VEL
LIN {X 0,Y 263.752,Z 372.627,A -85,B 0,C 180,E1 -18358.473,E2 -18358.473} C_VEL
LIN {X 0,Y 263.751,Z 372.628,A -85,B 0,C 180,E1 -18361.527,E2 -18361.527} C_VEL
LIN {X 0,Y 263.569,Z 372.655,A -85,B 0,C 180,E1 -18367.661,E2 -18367.661} C_VEL
LIN {X 0,Y 263.37,Z 372.672,A -85,B 0,C 180,E1 -18370.765,E2 -18370.765} C_VEL
LIN {X 0,Y 263.347,Z 372.681,A -85,B 0,C 180,E1 -18375.478,E2 -18375.478} C_VEL
LIN {X 0,Y 263.259,Z 372.689,A -85,B 0,C 180,E1 -18380.307,E2 -18380.307} C_VEL
LIN {X 0,Y 263.204,Z 372.704,A -85,B 0,C 180,E1 -18385.291,E2 -18385.291} C_VEL
LIN {X 0,Y 263.167,Z 372.705,A -85,B 0,C 180,E1 -18386.198,E2 -18386.198} C_VEL
LIN {X 0,Y 262.485,Z 372.793,A -85,B 0,C 180,E1 -18387.047,E2 -18387.047} C_VEL
LIN {X 0,Y 259.628,Z 373.149,A -85,B 0,C 180,E1 -18388.378,E2 -18388.378} C_VEL
LIN {X 0,Y 256.747,Z 373.507,A -85,B 0,C 180,E1 -18389.737,E2 -18389.737} C_VEL
LIN {X 0,Y 256.066,Z 373.588,A -85,B 0,C 180,E1 -18390.619,E2 -18390.619} C_VEL
LIN {X 0,Y 256.12,Z 373.744,A -85,B 0,C 180,E1 -18392.85,E2 -18392.85} C_VEL
LIN {X 0,Y 257.235,Z 378.704,A -85,B 0,C 180,E1 -18396.946,E2 -18396.946} C_VEL
LIN {X 0,Y 258.257,Z 383.805,A -85,B 0,C 180,E1 -18400.777,E2 -18400.777} C_VEL
LIN {X 0,Y 259.513,Z 390.316,A -85,B 0,C 180,E1 -18405.243,E2 -18405.243} C_VEL
LIN {X 0,Y 260.785,Z 397.35,A -85,B 0,C 180,E1 -18409.702,E2 -18409.702} C_VEL
LIN {X 0,Y 260.96,Z 400.161,A -85,B 0,C 180,E1 -18411.353,E2 -18411.353} C_VEL
LIN {X 0,Y 259.287,Z 407.421,A -85,B 0,C 180,E1 -18415.306,E2 -18415.306} C_VEL
LIN {X 0,Y 258.063,Z 413.25,A -85,B 0,C 180,E1 -18418.41,E2 -18418.41} C_VEL
LIN {X 0,Y 259.618,Z 419.994,A -85,B 0,C 180,E1 -18418.947,E2 -18418.947} C_VEL
LIN {X 0,Y 262.249,Z 432.525,A -85,B 0,C 180,E1 -18420.11,E2 -18420.11} C_VEL
LIN {X 0,Y 263.99,Z 445.28,A -85,B 0,C 180,E1 -18421.466,E2 -18421.466} C_VEL
LIN {X 0,Y 264.795,Z 457.026,A -85,B 0,C 180,E1 -18422.924,E2 -18422.924} C_VEL
LIN {X 0,Y 264.801,Z 468.94,A -85,B 0,C 180,E1 -18424.655,E2 -18424.655} C_VEL
LIN {X 0,Y 263.926,Z 479.562,A -85,B 0,C 180,E1 -18426.459,E2 -18426.459} C_VEL
LIN {X 0,Y 262.563,Z 487.334,A -85,B 0,C 180,E1 -18427.993,E2 -18427.993} C_VEL
LIN {X 0,Y 260.321,Z 495.482,A -85,B 0,C 180,E1 -18429.867,E2 -18429.867} C_VEL
LIN {X 0,Y 258.443,Z 502.543,A -85,B 0,C 180,E1 -18431.86,E2 -18431.86} C_VEL
LIN {X 0,Y 256.962,Z 509.064,A -85,B 0,C 180,E1 -18434.128,E2 -18434.128} C_VEL
LIN {X 0,Y 255.663,Z 514.505,A -85,B 0,C 180,E1 -18436.489,E2 -18436.489} C_VEL
LIN {X 0,Y 254.899,Z 518.805,A -85,B 0,C 180,E1 -18438.873,E2 -18438.873} C_VEL
LIN {X 0,Y 254.692,Z 521.113,A -85,B 0,C 180,E1 -18440.471,E2 -18440.471} C_VEL
LIN {X 0,Y 254.755,Z 524.397,A -85,B 0,C 180,E1 -18443.666,E2 -18443.666} C_VEL
LIN {X 0,Y 254.928,Z 525.438,A -85,B 0,C 180,E1 -18445.257,E2 -18445.257} C_VEL
LIN {X 0,Y 255.234,Z 526.075,A -85,B 0,C 180,E1 -18446.844,E2 -18446.844} C_VEL
LIN {X 0,Y 255.343,Z 526.243,A -85,B 0,C 180,E1 -18448.424,E2 -18448.424} C_VEL
LIN {X 0,Y 255.464,Z 526.007,A -85,B 0,C 180,E1 -18450.001,E2 -18450.001} C_VEL
LIN {X 0,Y 255.401,Z 525.341,A -85,B 0,C 180,E1 -18451.578,E2 -18451.578} C_VEL
LIN {X 0,Y 255.38,Z 524.257,A -85,B 0,C 180,E1 -18453.156,E2 -18453.156} C_VEL
LIN {X 0,Y 255.016,Z 521.724,A -85,B 0,C 180,E1 -18455.536,E2 -18455.536} C_VEL
LIN {X 0,Y 254.841,Z 518.146,A -85,B 0,C 180,E1 -18457.927,E2 -18457.927} C_VEL
LIN {X 0,Y 254.911,Z 513.441,A -85,B 0,C 180,E1 -18460.325,E2 -18460.325} C_VEL
LIN {X 0,Y 255.548,Z 506.34,A -85,B 0,C 180,E1 -18463.115,E2 -18463.115} C_VEL
LIN {X 0,Y 256.491,Z 498.656,A -85,B 0,C 180,E1 -18465.496,E2 -18465.496} C_VEL
LIN {X 0,Y 257.762,Z 490.863,A -85,B 0,C 180,E1 -18467.454,E2 -18467.454} C_VEL
LIN {X 0,Y 259.275,Z 481.396,A -85,B 0,C 180,E1 -18469.395,E2 -18469.395} C_VEL
LIN {X 0,Y 259.654,Z 471.946,A -85,B 0,C 180,E1 -18471.018,E2 -18471.018} C_VEL
LIN {X 0,Y 259.7,Z 459.393,A -85,B 0,C 180,E1 -18472.781,E2 -18472.781} C_VEL
LIN {X 0,Y 259.462,Z 447.583,A -85,B 0,C 180,E1 -18474.106,E2 -18474.106} C_VEL
LIN {X 0,Y 258.711,Z 436.507,A -85,B 0,C 180,E1 -18475.11,E2 -18475.11} C_VEL
LIN {X 0,Y 257.207,Z 423.778,A -85,B 0,C 180,E1 -18476.02,E2 -18476.02} C_VEL
LIN {X 0,Y 255.938,Z 415.49,A -85,B 0,C 180,E1 -18476.503,E2 -18476.503} C_VEL
LIN {X 0,Y 256.956,Z 407.86,A -85,B 0,C 180,E1 -18480.399,E2 -18480.399} C_VEL
LIN {X 0,Y 258.388,Z 399.205,A -85,B 0,C 180,E1 -18484.834,E2 -18484.834} C_VEL
LIN {X 0,Y 259.47,Z 392.762,A -85,B 0,C 180,E1 -18488.234,E2 -18488.234} C_VEL
LIN {X 0,Y 258.957,Z 388.446,A -85,B 0,C 180,E1 -18490.645,E2 -18490.645} C_VEL
LIN {X 0,Y 257.942,Z 383.047,A -85,B 0,C 180,E1 -18493.852,E2 -18493.852} C_VEL
LIN {X 0,Y 256.798,Z 377.018,A -85,B 0,C 180,E1 -18497.642,E2 -18497.642} C_VEL
LIN {X 0,Y 256.092,Z 373.585,A -85,B 0,C 180,E1 -18499.968,E2 -18499.968} C_VEL
LIN {X 0,Y 256.135,Z 373.583,A -85,B 0,C 180,E1 -18502.868,E2 -18502.868} C_VEL
LIN {X 0,Y 256.072,Z 373.59,A -85,B 0,C 180,E1 -18506.708,E2 -18506.708} C_VEL
LIN {X 0,Y 256.108,Z 373.584,A -85,B 0,C 180,E1 -18510.4,E2 -18510.4} C_VEL
LIN {X 0,Y 256.193,Z 373.576,A -85,B 0,C 180,E1 -18514.862,E2 -18514.862} C_VEL
LIN {X 0,Y 256.173,Z 373.577,A -85,B 0,C 180,E1 -18519.106,E2 -18519.106} C_VEL
LIN {X 0,Y 256.306,Z 373.56,A -85,B 0,C 180,E1 -18524.086,E2 -18524.086} C_VEL
LIN {X 0,Y 256.315,Z 373.557,A -85,B 0,C 180,E1 -18528.935,E2 -18528.935} C_VEL
LIN {X 0,Y 256.547,Z 373.529,A -85,B 0,C 180,E1 -18532.128,E2 -18532.128} C_VEL
LIN {X 0,Y 256.72,Z 373.5,A -85,B 0,C 180,E1 -18538.432,E2 -18538.432} C_VEL
LIN {X 0,Y 256.72,Z 373.504,A -85,B 0,C 180,E1 -18541.569,E2 -18541.569} C_VEL
LIN {X 0,Y 256.547,Z 373.521,A -85,B 0,C 180,E1 -18547.873,E2 -18547.873} C_VEL
LIN {X 0,Y 256.316,Z 373.555,A -85,B 0,C 180,E1 -18551.066,E2 -18551.066} C_VEL
LIN {X 0,Y 256.306,Z 373.552,A -85,B 0,C 180,E1 -18555.915,E2 -18555.915} C_VEL
LIN {X 0,Y 256.176,Z 373.571,A -85,B 0,C 180,E1 -18560.895,E2 -18560.895} C_VEL
LIN {X 0,Y 256.195,Z 373.569,A -85,B 0,C 180,E1 -18565.138,E2 -18565.138} C_VEL
LIN {X 0,Y 256.117,Z 373.578,A -85,B 0,C 180,E1 -18569.6,E2 -18569.6} C_VEL
LIN {X 0,Y 256.091,Z 373.585,A -85,B 0,C 180,E1 -18573.29,E2 -18573.29} C_VEL
LIN {X 0,Y 256.135,Z 373.58,A -85,B 0,C 180,E1 -18577.275,E2 -18577.275} C_VEL
LIN {X 0,Y 256.063,Z 373.589,A -85,B 0,C 180,E1 -18581.202,E2 -18581.202} C_VEL
LIN {X 0,Y 256.068,Z 373.588,A -85,B 0,C 180,E1 -18585.529,E2 -18585.529} C_VEL
LIN {X 0,Y 256.061,Z 373.587,A -85,B 0,C 180,E1 -18588.796,E2 -18588.796} C_VEL
LIN {X 0,Y 256.137,Z 373.578,A -85,B 0,C 180,E1 -18592.867,E2 -18592.867} C_VEL
LIN {X 0,Y 256.074,Z 373.587,A -85,B 0,C 180,E1 -18596.707,E2 -18596.707} C_VEL
LIN {X 0,Y 256.12,Z 373.581,A -85,B 0,C 180,E1 -18600.4,E2 -18600.4} C_VEL
LIN {X 0,Y 256.194,Z 373.574,A -85,B 0,C 180,E1 -18604.861,E2 -18604.861} C_VEL
LIN {X 0,Y 256.173,Z 373.577,A -85,B 0,C 180,E1 -18609.104,E2 -18609.104} C_VEL
LIN {X 0,Y 256.237,Z 373.683,A -85,B 0,C 180,E1 -18612.484,E2 -18612.484} C_VEL
LIN {X 0,Y 260.671,Z 385.693,A -85,B 0,C 180,E1 -18613.903,E2 -18613.903} C_VEL
LIN {X 0,Y 264.215,Z 397.177,A -85,B 0,C 180,E1 -18615.49,E2 -18615.49} C_VEL
LIN {X 0,Y 265.214,Z 401.91,A -85,B 0,C 180,E1 -18616.201,E2 -18616.201} C_VEL
LIN {X 0,Y 263.678,Z 413.536,A -85,B 0,C 180,E1 -18617.883,E2 -18617.883} C_VEL
LIN {X 0,Y 262.383,Z 422.884,A -85,B 0,C 180,E1 -18619.582,E2 -18619.582} C_VEL
LIN {X 0,Y 261.012,Z 431.439,A -85,B 0,C 180,E1 -18621.482,E2 -18621.482} C_VEL
LIN {X 0,Y 259.487,Z 439.781,A -85,B 0,C 180,E1 -18623.779,E2 -18623.779} C_VEL
LIN {X 0,Y 258.251,Z 446.48,A -85,B 0,C 180,E1 -18626.098,E2 -18626.098} C_VEL
LIN {X 0,Y 257.332,Z 451.838,A -85,B 0,C 180,E1 -18628.434,E2 -18628.434} C_VEL
LIN {X 0,Y 256.603,Z 456.051,A -85,B 0,C 180,E1 -18630.784,E2 -18630.784} C_VEL
LIN {X 0,Y 256.04,Z 459.238,A -85,B 0,C 180,E1 -18633.146,E2 -18633.146} C_VEL
LIN {X 0,Y 255.974,Z 460.81,A -85,B 0,C 180,E1 -18634.724,E2 -18634.724} C_VEL
LIN {X 0,Y 255.958,Z 461.989,A -85,B 0,C 180,E1 -18636.304,E2 -18636.304} C_VEL
LIN {X 0,Y 256.029,Z 463.131,A -85,B 0,C 180,E1 -18639.479,E2 -18639.479} C_VEL
LIN {X 0,Y 256.252,Z 463.133,A -85,B 0,C 180,E1 -18641.067,E2 -18641.067} C_VEL
LIN {X 0,Y 256.555,Z 462.748,A -85,B 0,C 180,E1 -18642.658,E2 -18642.658} C_VEL
LIN {X 0,Y 257.516,Z 460.715,A -85,B 0,C 180,E1 -18645.837,E2 -18645.837} C_VEL
LIN {X 0,Y 258.498,Z 458.492,A -85,B 0,C 180,E1 -18647.902,E2 -18647.902} C_VEL
LIN {X 0,Y 259.992,Z 454.447,A -85,B 0,C 180,E1 -18650.572,E2 -18650.572} C_VEL
LIN {X 0,Y 261.622,Z 449.658,A -85,B 0,C 180,E1 -18652.923,E2 -18652.923} C_VEL
LIN {X 0,Y 263.592,Z 443.566,A -85,B 0,C 180,E1 -18655.251,E2 -18655.251} C_VEL
LIN {X 0,Y 265.91,Z 435.893,A -85,B 0,C 180,E1 -18657.549,E2 -18657.549} C_VEL
LIN {X 0,Y 267.989,Z 427.982,A -85,B 0,C 180,E1 -18659.452,E2 -18659.452} C_VEL
LIN {X 0,Y 270.215,Z 418.262,A -85,B 0,C 180,E1 -18661.343,E2 -18661.343} C_VEL
LIN {X 0,Y 271.405,Z 412.655,A -85,B 0,C 180,E1 -18662.257,E2 -18662.257} C_VEL
LIN {X 0,Y 269.031,Z 404.18,A -85,B 0,C 180,E1 -18663.982,E2 -18663.982} C_VEL
LIN {X 0,Y 265.708,Z 394.65,A -85,B 0,C 180,E1 -18665.772,E2 -18665.772} C_VEL
LIN {X 0,Y 261.394,Z 384.529,A -85,B 0,C 180,E1 -18667.544,E2 -18667.544} C_VEL
LIN {X 0,Y 257.315,Z 376.725,A -85,B 0,C 180,E1 -18668.871,E2 -18668.871} C_VEL
LIN {X 0,Y 256.118,Z 373.913,A -85,B 0,C 180,E1 -18669.28,E2 -18669.28} C_VEL
LIN {X 0,Y 256.066,Z 373.589,A -85,B 0,C 180,E1 -18669.395,E2 -18669.395} C_VEL
LIN {X 0,Y 256.061,Z 373.591,A -85,B 0,C 180,E1 -18673.326,E2 -18673.326} C_VEL
LIN {X 0,Y 256.086,Z 373.587,A -85,B 0,C 180,E1 -18677.814,E2 -18677.814} C_VEL
LIN {X 0,Y 256.104,Z 373.583,A -85,B 0,C 180,E1 -18680.863,E2 -18680.863} C_VEL
LIN {X 0,Y 256.12,Z 373.581,A -85,B 0,C 180,E1 -18684.812,E2 -18684.812} C_VEL
LIN {X 0,Y 256.091,Z 373.55,A -85,B 0,C 180,E1 -18688.572,E2 -18688.572} C_VEL
LIN {X 0,Y 256.136,Z 373.56,A -85,B 0,C 180,E1 -18692.195,E2 -18692.195} C_VEL
LIN {X 0,Y 256.164,Z 373.57,A -85,B 0,C 180,E1 -18695.698,E2 -18695.698} C_VEL
LIN {X 0,Y 256.164,Z 373.575,A -85,B 0,C 180,E1 -18699.104,E2 -18699.104} C_VEL
LIN {X 0,Y 256.297,Z 373.558,A -85,B 0,C 180,E1 -18704.084,E2 -18704.084} C_VEL
LIN {X 0,Y 256.307,Z 373.559,A -85,B 0,C 180,E1 -18708.933,E2 -18708.933} C_VEL
LIN {X 0,Y 256.537,Z 373.529,A -85,B 0,C 180,E1 -18712.127,E2 -18712.127} C_VEL
LIN {X 0,Y 256.714,Z 373.504,A -85,B 0,C 180,E1 -18718.431,E2 -18718.431} C_VEL
LIN {X 0,Y 256.714,Z 373.505,A -85,B 0,C 180,E1 -18721.568,E2 -18721.568} C_VEL
LIN {X 0,Y 256.536,Z 373.531,A -85,B 0,C 180,E1 -18727.873,E2 -18727.873} C_VEL
LIN {X 0,Y 256.306,Z 373.555,A -85,B 0,C 180,E1 -18731.066,E2 -18731.066} C_VEL
LIN {X 0,Y 256.296,Z 373.561,A -85,B 0,C 180,E1 -18735.915,E2 -18735.915} C_VEL
LIN {X 0,Y 256.162,Z 373.572,A -85,B 0,C 180,E1 -18740.895,E2 -18740.895} C_VEL
LIN {X 0,Y 256.184,Z 373.579,A -85,B 0,C 180,E1 -18745.139,E2 -18745.139} C_VEL
LIN {X 0,Y 256.11,Z 373.586,A -85,B 0,C 180,E1 -18749.6,E2 -18749.6} C_VEL
LIN {X 0,Y 256.066,Z 373.588,A -85,B 0,C 180,E1 -18750.619,E2 -18750.619} C_VEL
LIN {X 0,Y 255.496,Z 374.058,A -85,B 0,C 180,E1 -18751.926,E2 -18751.926} C_VEL
LIN {X 0,Y 254.169,Z 375.251,A -85,B 0,C 180,E1 -18753.199,E2 -18753.199} C_VEL
LIN {X 0,Y 251.182,Z 378.791,A -85,B 0,C 180,E1 -18755.716,E2 -18755.716} C_VEL
LIN {X 0,Y 250.497,Z 380.667,A -85,B 0,C 180,E1 -18757.01,E2 -18757.01} C_VEL
LIN {X 0,Y 250.516,Z 381.246,A -85,B 0,C 180,E1 -18757.448,E2 -18757.448} C_VEL
LIN {X 0,Y 251.434,Z 385.894,A -85,B 0,C 180,E1 -18761.003,E2 -18761.003} C_VEL
LIN {X 0,Y 252.55,Z 391.642,A -85,B 0,C 180,E1 -18765.055,E2 -18765.055} C_VEL
LIN {X 0,Y 253.767,Z 398.412,A -85,B 0,C 180,E1 -18769.491,E2 -18769.491} C_VEL
LIN {X 0,Y 254.018,Z 400.494,A -85,B 0,C 180,E1 -18770.776,E2 -18770.776} C_VEL
LIN {X 0,Y 253.482,Z 403.357,A -85,B 0,C 180,E1 -18772.414,E2 -18772.414} C_VEL
LIN {X 0,Y 251.539,Z 411.543,A -85,B 0,C 180,E1 -18776.95,E2 -18776.95} C_VEL
LIN {X 0,Y 251.391,Z 412.247,A -85,B 0,C 180,E1 -18777.337,E2 -18777.337} C_VEL
LIN {X 0,Y 252.259,Z 416.019,A -85,B 0,C 180,E1 -18777.64,E2 -18777.64} C_VEL
LIN {X 0,Y 255.415,Z 430.103,A -85,B 0,C 180,E1 -18778.992,E2 -18778.992} C_VEL
LIN {X 0,Y 257.325,Z 443.357,A -85,B 0,C 180,E1 -18780.443,E2 -18780.443} C_VEL
LIN {X 0,Y 258.172,Z 455.253,A -85,B 0,C 180,E1 -18781.946,E2 -18781.946} C_VEL
LIN {X 0,Y 258.272,Z 466.087,A -85,B 0,C 180,E1 -18783.541,E2 -18783.541} C_VEL
LIN {X 0,Y 257.65,Z 475.907,A -85,B 0,C 180,E1 -18785.205,E2 -18785.205} C_VEL
LIN {X 0,Y 256.381,Z 485.052,A -85,B 0,C 180,E1 -18787.008,E2 -18787.008} C_VEL
LIN {X 0,Y 254.067,Z 493.428,A -85,B 0,C 180,E1 -18788.925,E2 -18788.925} C_VEL
LIN {X 0,Y 251.739,Z 501.687,A -85,B 0,C 180,E1 -18791.275,E2 -18791.275} C_VEL
LIN {X 0,Y 250.406,Z 507.002,A -85,B 0,C 180,E1 -18793.135,E2 -18793.135} C_VEL
LIN {X 0,Y 248.688,Z 513.799,A -85,B 0,C 180,E1 -18796.102,E2 -18796.102} C_VEL
LIN {X 0,Y 247.876,Z 518.059,A -85,B 0,C 180,E1 -18798.554,E2 -18798.554} C_VEL
LIN {X 0,Y 247.62,Z 520.326,A -85,B 0,C 180,E1 -18800.196,E2 -18800.196} C_VEL
LIN {X 0,Y 247.669,Z 523.577,A -85,B 0,C 180,E1 -18803.484,E2 -18803.484} C_VEL
LIN {X 0,Y 247.836,Z 524.602,A -85,B 0,C 180,E1 -18805.121,E2 -18805.121} C_VEL
LIN {X 0,Y 248.149,Z 525.205,A -85,B 0,C 180,E1 -18806.754,E2 -18806.754} C_VEL
LIN {X 0,Y 248.294,Z 525.36,A -85,B 0,C 180,E1 -18808.379,E2 -18808.379} C_VEL
LIN {X 0,Y 248.418,Z 525.108,A -85,B 0,C 180,E1 -18810.001,E2 -18810.001} C_VEL
LIN {X 0,Y 248.354,Z 524.424,A -85,B 0,C 180,E1 -18811.623,E2 -18811.623} C_VEL
LIN {X 0,Y 248.311,Z 523.3,A -85,B 0,C 180,E1 -18813.246,E2 -18813.246} C_VEL
LIN {X 0,Y 247.942,Z 520.734,A -85,B 0,C 180,E1 -18815.695,E2 -18815.695} C_VEL
LIN {X 0,Y 247.775,Z 517.115,A -85,B 0,C 180,E1 -18818.154,E2 -18818.154} C_VEL
LIN {X 0,Y 247.857,Z 512.357,A -85,B 0,C 180,E1 -18820.622,E2 -18820.622} C_VEL
LIN {X 0,Y 248.43,Z 506.346,A -85,B 0,C 180,E1 -18823.082,E2 -18823.082} C_VEL
LIN {X 0,Y 249.372,Z 498.848,A -85,B 0,C 180,E1 -18825.531,E2 -18825.531} C_VEL
LIN {X 0,Y 250.527,Z 491.758,A -85,B 0,C 180,E1 -18827.427,E2 -18827.427} C_VEL
LIN {X 0,Y 252.134,Z 482.075,A -85,B 0,C 180,E1 -18829.543,E2 -18829.543} C_VEL
LIN {X 0,Y 252.62,Z 474.211,A -85,B 0,C 180,E1 -18830.99,E2 -18830.99} C_VEL
LIN {X 0,Y 252.81,Z 463.299,A -85,B 0,C 180,E1 -18832.69,E2 -18832.69} C_VEL
LIN {X 0,Y 252.778,Z 452.192,A -85,B 0,C 180,E1 -18834.099,E2 -18834.099} C_VEL
LIN {X 0,Y 252.177,Z 439.694,A -85,B 0,C 180,E1 -18835.375,E2 -18835.375} C_VEL
LIN {X 0,Y 250.852,Z 427.095,A -85,B 0,C 180,E1 -18836.394,E2 -18836.394} C_VEL
LIN {X 0,Y 249.007,Z 414.565,A -85,B 0,C 180,E1 -18837.187,E2 -18837.187} C_VEL
LIN {X 0,Y 250.143,Z 406.767,A -85,B 0,C 180,E1 -18841.318,E2 -18841.318} C_VEL
LIN {X 0,Y 251.692,Z 398.108,A -85,B 0,C 180,E1 -18845.927,E2 -18845.927} C_VEL
LIN {X 0,Y 252.331,Z 394.655,A -85,B 0,C 180,E1 -18847.79,E2 -18847.79} C_VEL
LIN {X 0,Y 252.442,Z 392.885,A -85,B 0,C 180,E1 -18848.783,E2 -18848.783} C_VEL
LIN {X 0,Y 251.553,Z 387.22,A -85,B 0,C 180,E1 -18852.109,E2 -18852.109} C_VEL
LIN {X 0,Y 250.083,Z 379.587,A -85,B 0,C 180,E1 -18856.944,E2 -18856.944} C_VEL
LIN {X 0,Y 249.047,Z 374.464,A -85,B 0,C 180,E1 -18860.454,E2 -18860.454} C_VEL
LIN {X 0,Y 249.049,Z 374.467,A -85,B 0,C 180,E1 -18864.923,E2 -18864.923} C_VEL
LIN {X 0,Y 249.052,Z 374.462,A -85,B 0,C 180,E1 -18869.473,E2 -18869.473} C_VEL
LIN {X 0,Y 249.077,Z 374.46,A -85,B 0,C 180,E1 -18873.163,E2 -18873.163} C_VEL
LIN {X 0,Y 249.085,Z 374.462,A -85,B 0,C 180,E1 -18876.733,E2 -18876.733} C_VEL
LIN {X 0,Y 249.117,Z 374.457,A -85,B 0,C 180,E1 -18880.212,E2 -18880.212} C_VEL
LIN {X 0,Y 249.247,Z 374.438,A -85,B 0,C 180,E1 -18883.623,E2 -18883.623} C_VEL
LIN {X 0,Y 249.259,Z 374.438,A -85,B 0,C 180,E1 -18888.617,E2 -18888.617} C_VEL
LIN {X 0,Y 249.491,Z 374.407,A -85,B 0,C 180,E1 -18891.903,E2 -18891.903} C_VEL
LIN {X 0,Y 249.441,Z 374.408,A -85,B 0,C 180,E1 -18896.77,E2 -18896.77} C_VEL
LIN {X 0,Y 249.735,Z 374.371,A -85,B 0,C 180,E1 -18900,E2 -18900} C_VEL
LIN {X 0,Y 249.441,Z 374.411,A -85,B 0,C 180,E1 -18903.231,E2 -18903.231} C_VEL
LIN {X 0,Y 249.491,Z 374.401,A -85,B 0,C 180,E1 -18908.097,E2 -18908.097} C_VEL
LIN {X 0,Y 249.259,Z 374.434,A -85,B 0,C 180,E1 -18911.384,E2 -18911.384} C_VEL
LIN {X 0,Y 249.248,Z 374.434,A -85,B 0,C 180,E1 -18916.378,E2 -18916.378} C_VEL
LIN {X 0,Y 249.094,Z 374.455,A -85,B 0,C 180,E1 -18921.518,E2 -18921.518} C_VEL
LIN {X 0,Y 249.137,Z 374.45,A -85,B 0,C 180,E1 -18925.482,E2 -18925.482} C_VEL
LIN {X 0,Y 249.087,Z 374.454,A -85,B 0,C 180,E1 -18928.992,E2 -18928.992} C_VEL
LIN {X 0,Y 249.042,Z 374.461,A -85,B 0,C 180,E1 -18932.425,E2 -18932.425} C_VEL
LIN {X 0,Y 249.075,Z 374.457,A -85,B 0,C 180,E1 -18936.338,E2 -18936.338} C_VEL
LIN {X 0,Y 249.032,Z 374.462,A -85,B 0,C 180,E1 -18940.474,E2 -18940.474} C_VEL
LIN {X 0,Y 249.013,Z 374.464,A -85,B 0,C 180,E1 -18944.878,E2 -18944.878} C_VEL
LIN {X 0,Y 249.024,Z 374.464,A -85,B 0,C 180,E1 -18947.363,E2 -18947.363} C_VEL
LIN {X 0,Y 249.05,Z 374.458,A -85,B 0,C 180,E1 -18952.2,E2 -18952.2} C_VEL
LIN {X 0,Y 249.049,Z 374.461,A -85,B 0,C 180,E1 -18955.639,E2 -18955.639} C_VEL
LIN {X 0,Y 249.058,Z 374.462,A -85,B 0,C 180,E1 -18959.473,E2 -18959.473} C_VEL
LIN {X 0,Y 249.08,Z 374.461,A -85,B 0,C 180,E1 -18963.162,E2 -18963.162} C_VEL
LIN {X 0,Y 249.086,Z 374.459,A -85,B 0,C 180,E1 -18966.732,E2 -18966.732} C_VEL
LIN {X 0,Y 249.144,Z 374.452,A -85,B 0,C 180,E1 -18971.496,E2 -18971.496} C_VEL
LIN {X 0,Y 249.163,Z 374.632,A -85,B 0,C 180,E1 -18971.817,E2 -18971.817} C_VEL
LIN {X 0,Y 253.752,Z 386.663,A -85,B 0,C 180,E1 -18973.313,E2 -18973.313} C_VEL
LIN {X 0,Y 257.002,Z 397.192,A -85,B 0,C 180,E1 -18974.812,E2 -18974.812} C_VEL
LIN {X 0,Y 258.432,Z 402.572,A -85,B 0,C 180,E1 -18975.663,E2 -18975.663} C_VEL
LIN {X 0,Y 257.181,Z 412.869,A -85,B 0,C 180,E1 -18977.17,E2 -18977.17} C_VEL
LIN {X 0,Y 255.782,Z 422.482,A -85,B 0,C 180,E1 -18978.91,E2 -18978.91} C_VEL
LIN {X 0,Y 254.339,Z 431.247,A -85,B 0,C 180,E1 -18980.857,E2 -18980.857} C_VEL
LIN {X 0,Y 252.747,Z 439.833,A -85,B 0,C 180,E1 -18983.212,E2 -18983.212} C_VEL
LIN {X 0,Y 251.408,Z 446.693,A -85,B 0,C 180,E1 -18985.59,E2 -18985.59} C_VEL
LIN {X 0,Y 250.299,Z 452.974,A -85,B 0,C 180,E1 -18988.39,E2 -18988.39} C_VEL
LIN {X 0,Y 249.544,Z 457.13,A -85,B 0,C 180,E1 -18990.806,E2 -18990.806} C_VEL
LIN {X 0,Y 248.985,Z 460.259,A -85,B 0,C 180,E1 -18993.235,E2 -18993.235} C_VEL
LIN {X 0,Y 248.934,Z 461.803,A -85,B 0,C 180,E1 -18994.857,E2 -18994.857} C_VEL
LIN {X 0,Y 248.915,Z 462.934,A -85,B 0,C 180,E1 -18996.484,E2 -18996.484} C_VEL
LIN {X 0,Y 249.019,Z 464.022,A -85,B 0,C 180,E1 -18999.748,E2 -18999.748} C_VEL
LIN {X 0,Y 249.257,Z 464,A -85,B 0,C 180,E1 -19001.382,E2 -19001.382} C_VEL
LIN {X 0,Y 249.593,Z 463.563,A -85,B 0,C 180,E1 -19003.017,E2 -19003.017} C_VEL
LIN {X 0,Y 250.66,Z 461.474,A -85,B 0,C 180,E1 -19006.282,E2 -19006.282} C_VEL
LIN {X 0,Y 251.639,Z 459.364,A -85,B 0,C 180,E1 -19008.269,E2 -19008.269} C_VEL
LIN {X 0,Y 253.28,Z 455.094,A -85,B 0,C 180,E1 -19011.143,E2 -19011.143} C_VEL
LIN {X 0,Y 255.044,Z 450.238,A -85,B 0,C 180,E1 -19013.55,E2 -19013.55} C_VEL
LIN {X 0,Y 257.119,Z 444.077,A -85,B 0,C 180,E1 -19015.933,E2 -19015.933} C_VEL
LIN {X 0,Y 259.577,Z 436.281,A -85,B 0,C 180,E1 -19018.281,E2 -19018.281} C_VEL
LIN {X 0,Y 261.747,Z 428.272,A -85,B 0,C 180,E1 -19020.227,E2 -19020.227} C_VEL
LIN {X 0,Y 264.108,Z 418.43,A -85,B 0,C 180,E1 -19022.153,E2 -19022.153} C_VEL
LIN {X 0,Y 264.932,Z 414.681,A -85,B 0,C 180,E1 -19022.774,E2 -19022.774} C_VEL
LIN {X 0,Y 262.356,Z 405.391,A -85,B 0,C 180,E1 -19024.76,E2 -19024.76} C_VEL
LIN {X 0,Y 258.949,Z 395.76,A -85,B 0,C 180,E1 -19026.66,E2 -19026.66} C_VEL
LIN {X 0,Y 254.852,Z 386.406,A -85,B 0,C 180,E1 -19028.405,E2 -19028.405} C_VEL
LIN {X 0,Y 250.53,Z 378.049,A -85,B 0,C 180,E1 -19029.908,E2 -19029.908} C_VEL
LIN {X 0,Y 249.234,Z 375.569,A -85,B 0,C 180,E1 -19030.337,E2 -19030.337} C_VEL
LIN {X 0,Y 248.993,Z 374.469,A -85,B 0,C 180,E1 -19030.479,E2 -19030.479} C_VEL
LIN {X 0,Y 249.008,Z 374.468,A -85,B 0,C 180,E1 -19032.791,E2 -19032.791} C_VEL
LIN {X 0,Y 249.026,Z 374.464,A -85,B 0,C 180,E1 -19037.364,E2 -19037.364} C_VEL
LIN {X 0,Y 249.05,Z 374.466,A -85,B 0,C 180,E1 -19041.623,E2 -19041.623} C_VEL
LIN {X 0,Y 249.06,Z 374.463,A -85,B 0,C 180,E1 -19045.641,E2 -19045.641} C_VEL
LIN {X 0,Y 249.046,Z 374.419,A -85,B 0,C 180,E1 -19049.472,E2 -19049.472} C_VEL
LIN {X 0,Y 249.07,Z 374.452,A -85,B 0,C 180,E1 -19053.161,E2 -19053.161} C_VEL
LIN {X 0,Y 249.076,Z 374.445,A -85,B 0,C 180,E1 -19056.732,E2 -19056.732} C_VEL
LIN {X 0,Y 249.108,Z 374.454,A -85,B 0,C 180,E1 -19060.211,E2 -19060.211} C_VEL
LIN {X 0,Y 249.239,Z 374.433,A -85,B 0,C 180,E1 -19063.621,E2 -19063.621} C_VEL
LIN {X 0,Y 249.25,Z 374.438,A -85,B 0,C 180,E1 -19068.616,E2 -19068.616} C_VEL
LIN {X 0,Y 249.481,Z 374.409,A -85,B 0,C 180,E1 -19071.902,E2 -19071.902} C_VEL
LIN {X 0,Y 249.439,Z 374.414,A -85,B 0,C 180,E1 -19076.769,E2 -19076.769} C_VEL
LIN {X 0,Y 249.733,Z 374.363,A -85,B 0,C 180,E1 -19080,E2 -19080} C_VEL
LIN {X 0,Y 249.438,Z 374.414,A -85,B 0,C 180,E1 -19083.23,E2 -19083.23} C_VEL
LIN {X 0,Y 249.48,Z 374.408,A -85,B 0,C 180,E1 -19088.097,E2 -19088.097} C_VEL
LIN {X 0,Y 249.249,Z 374.436,A -85,B 0,C 180,E1 -19091.383,E2 -19091.383} C_VEL
LIN {X 0,Y 249.238,Z 374.438,A -85,B 0,C 180,E1 -19096.378,E2 -19096.378} C_VEL
LIN {X 0,Y 249.083,Z 374.456,A -85,B 0,C 180,E1 -19101.518,E2 -19101.518} C_VEL
LIN {X 0,Y 249.127,Z 374.457,A -85,B 0,C 180,E1 -19105.483,E2 -19105.483} C_VEL
LIN {X 0,Y 249.079,Z 374.464,A -85,B 0,C 180,E1 -19108.994,E2 -19108.994} C_VEL
LIN {X 0,Y 249.062,Z 374.569,A -85,B 0,C 180,E1 -19111.79,E2 -19111.79} C_VEL
LIN {X 0,Y 250.184,Z 379.623,A -85,B 0,C 180,E1 -19116.151,E2 -19116.151} C_VEL
LIN {X 0,Y 250.516,Z 381.246,A -85,B 0,C 180,E1 -19117.448,E2 -19117.448} C_VEL
LIN {X 0,Y 250.16,Z 383.074,A -85,B 0,C 180,E1 -19118.731,E2 -19118.731} C_VEL
LIN {X 0,Y 247.889,Z 386.518,A -85,B 0,C 180,E1 -19120.806,E2 -19120.806} C_VEL
LIN {X 0,Y 245.984,Z 389.365,A -85,B 0,C 180,E1 -19122.487,E2 -19122.487} C_VEL
LIN {X 0,Y 245.359,Z 391.396,A -85,B 0,C 180,E1 -19123.787,E2 -19123.787} C_VEL
LIN {X 0,Y 245.416,Z 392.03,A -85,B 0,C 180,E1 -19124.227,E2 -19124.227} C_VEL
LIN {X 0,Y 246.363,Z 397.376,A -85,B 0,C 180,E1 -19127.876,E2 -19127.876} C_VEL
LIN {X 0,Y 246.971,Z 400.941,A -85,B 0,C 180,E1 -19130.204,E2 -19130.204} C_VEL
LIN {X 0,Y 246.934,Z 402.601,A -85,B 0,C 180,E1 -19131.235,E2 -19131.235} C_VEL
LIN {X 0,Y 244.769,Z 411.219,A -85,B 0,C 180,E1 -19136.18,E2 -19136.18} C_VEL
LIN {X 0,Y 245.662,Z 415.076,A -85,B 0,C 180,E1 -19136.526,E2 -19136.526} C_VEL
LIN {X 0,Y 248.87,Z 429.397,A -85,B 0,C 180,E1 -19137.975,E2 -19137.975} C_VEL
LIN {X 0,Y 250.781,Z 442.437,A -85,B 0,C 180,E1 -19139.475,E2 -19139.475} C_VEL
LIN {X 0,Y 251.642,Z 454.177,A -85,B 0,C 180,E1 -19141.018,E2 -19141.018} C_VEL
LIN {X 0,Y 251.68,Z 465.801,A -85,B 0,C 180,E1 -19142.792,E2 -19142.792} C_VEL
LIN {X 0,Y 251.021,Z 475.715,A -85,B 0,C 180,E1 -19144.545,E2 -19144.545} C_VEL
LIN {X 0,Y 249.748,Z 484.58,A -85,B 0,C 180,E1 -19146.361,E2 -19146.361} C_VEL
LIN {X 0,Y 247.437,Z 492.893,A -85,B 0,C 180,E1 -19148.332,E2 -19148.332} C_VEL
LIN {X 0,Y 244.993,Z 501.088,A -85,B 0,C 180,E1 -19150.739,E2 -19150.739} C_VEL
LIN {X 0,Y 243.218,Z 507.751,A -85,B 0,C 180,E1 -19153.206,E2 -19153.206} C_VEL
LIN {X 0,Y 241.734,Z 513.091,A -85,B 0,C 180,E1 -19155.694,E2 -19155.694} C_VEL
LIN {X 0,Y 240.868,Z 517.312,A -85,B 0,C 180,E1 -19158.216,E2 -19158.216} C_VEL
LIN {X 0,Y 240.575,Z 519.541,A -85,B 0,C 180,E1 -19159.906,E2 -19159.906} C_VEL
LIN {X 0,Y 240.599,Z 522.759,A -85,B 0,C 180,E1 -19163.291,E2 -19163.291} C_VEL
LIN {X 0,Y 240.745,Z 523.762,A -85,B 0,C 180,E1 -19164.977,E2 -19164.977} C_VEL
LIN {X 0,Y 241.066,Z 524.335,A -85,B 0,C 180,E1 -19166.659,E2 -19166.659} C_VEL
LIN {X 0,Y 241.245,Z 524.477,A -85,B 0,C 180,E1 -19168.332,E2 -19168.332} C_VEL
LIN {X 0,Y 241.372,Z 524.208,A -85,B 0,C 180,E1 -19170.001,E2 -19170.001} C_VEL
LIN {X 0,Y 241.307,Z 523.505,A -85,B 0,C 180,E1 -19171.67,E2 -19171.67} C_VEL
LIN {X 0,Y 241.225,Z 522.339,A -85,B 0,C 180,E1 -19173.342,E2 -19173.342} C_VEL
LIN {X 0,Y 240.872,Z 519.736,A -85,B 0,C 180,E1 -19175.863,E2 -19175.863} C_VEL
LIN {X 0,Y 240.71,Z 516.075,A -85,B 0,C 180,E1 -19178.396,E2 -19178.396} C_VEL
LIN {X 0,Y 240.821,Z 511.266,A -85,B 0,C 180,E1 -19180.936,E2 -19180.936} C_VEL
LIN {X 0,Y 241.608,Z 504.053,A -85,B 0,C 180,E1 -19183.887,E2 -19183.887} C_VEL
LIN {X 0,Y 242.621,Z 496.245,A -85,B 0,C 180,E1 -19186.406,E2 -19186.406} C_VEL
LIN {X 0,Y 244.158,Z 488.335,A -85,B 0,C 180,E1 -19188.461,E2 -19188.461} C_VEL
LIN {X 0,Y 245.522,Z 478.58,A -85,B 0,C 180,E1 -19190.528,E2 -19190.528} C_VEL
LIN {X 0,Y 245.837,Z 467.506,A -85,B 0,C 180,E1 -19192.482,E2 -19192.482} C_VEL
LIN {X 0,Y 245.999,Z 456.632,A -85,B 0,C 180,E1 -19194.044,E2 -19194.044} C_VEL
LIN {X 0,Y 245.737,Z 444.998,A -85,B 0,C 180,E1 -19195.405,E2 -19195.405} C_VEL
LIN {X 0,Y 244.594,Z 431.181,A -85,B 0,C 180,E1 -19196.691,E2 -19196.691} C_VEL
LIN {X 0,Y 242.718,Z 418.035,A -85,B 0,C 180,E1 -19197.643,E2 -19197.643} C_VEL
LIN {X 0,Y 242.106,Z 413.709,A -85,B 0,C 180,E1 -19197.911,E2 -19197.911} C_VEL
LIN {X 0,Y 243.352,Z 405.671,A -85,B 0,C 180,E1 -19202.296,E2 -19202.296} C_VEL
LIN {X 0,Y 245.03,Z 397.024,A -85,B 0,C 180,E1 -19207.038,E2 -19207.038} C_VEL
LIN {X 0,Y 245.363,Z 393.521,A -85,B 0,C 180,E1 -19209.063,E2 -19209.063} C_VEL
LIN {X 0,Y 244.354,Z 387.421,A -85,B 0,C 180,E1 -19212.806,E2 -19212.806} C_VEL
LIN {X 0,Y 243.056,Z 380.615,A -85,B 0,C 180,E1 -19217.252,E2 -19217.252} C_VEL
LIN {X 0,Y 241.974,Z 375.345,A -85,B 0,C 180,E1 -19221.036,E2 -19221.036} C_VEL
LIN {X 0,Y 241.992,Z 375.345,A -85,B 0,C 180,E1 -19224.49,E2 -19224.49} C_VEL
LIN {X 0,Y 241.978,Z 375.344,A -85,B 0,C 180,E1 -19228.48,E2 -19228.48} C_VEL
LIN {X 0,Y 242.007,Z 375.34,A -85,B 0,C 180,E1 -19232.313,E2 -19232.313} C_VEL
LIN {X 0,Y 242.062,Z 375.334,A -85,B 0,C 180,E1 -19236.017,E2 -19236.017} C_VEL
LIN {X 0,Y 242.043,Z 375.336,A -85,B 0,C 180,E1 -19239.609,E2 -19239.609} C_VEL
LIN {X 0,Y 242.169,Z 375.32,A -85,B 0,C 180,E1 -19243.279,E2 -19243.279} C_VEL
LIN {X 0,Y 242.192,Z 375.318,A -85,B 0,C 180,E1 -19248.28,E2 -19248.28} C_VEL
LIN {X 0,Y 242.441,Z 375.284,A -85,B 0,C 180,E1 -19251.666,E2 -19251.666} C_VEL
LIN {X 0,Y 242.265,Z 375.305,A -85,B 0,C 180,E1 -19255.008,E2 -19255.008} C_VEL
LIN {X 0,Y 242.642,Z 375.252,A -85,B 0,C 180,E1 -19258.341,E2 -19258.341} C_VEL
LIN {X 0,Y 242.642,Z 375.258,A -85,B 0,C 180,E1 -19261.66,E2 -19261.66} C_VEL
LIN {X 0,Y 242.435,Z 375.275,A -85,B 0,C 180,E1 -19266.756,E2 -19266.756} C_VEL
LIN {X 0,Y 242.352,Z 375.296,A -85,B 0,C 180,E1 -19270.021,E2 -19270.021} C_VEL
LIN {X 0,Y 242.173,Z 375.308,A -85,B 0,C 180,E1 -19275.141,E2 -19275.141} C_VEL
LIN {X 0,Y 242.08,Z 375.328,A -85,B 0,C 180,E1 -19278.624,E2 -19278.624} C_VEL
LIN {X 0,Y 242.02,Z 375.33,A -85,B 0,C 180,E1 -19282.18,E2 -19282.18} C_VEL
LIN {X 0,Y 242.073,Z 375.333,A -85,B 0,C 180,E1 -19285.838,E2 -19285.838} C_VEL
LIN {X 0,Y 242.035,Z 375.331,A -85,B 0,C 180,E1 -19289.58,E2 -19289.58} C_VEL
LIN {X 0,Y 241.998,Z 375.342,A -85,B 0,C 180,E1 -19293.491,E2 -19293.491} C_VEL
LIN {X 0,Y 242.009,Z 375.339,A -85,B 0,C 180,E1 -19297.579,E2 -19297.579} C_VEL
LIN {X 0,Y 241.95,Z 375.344,A -85,B 0,C 180,E1 -19301.92,E2 -19301.92} C_VEL
LIN {X 0,Y 241.943,Z 375.344,A -85,B 0,C 180,E1 -19306.57,E2 -19306.57} C_VEL
LIN {X 0,Y 241.962,Z 375.341,A -85,B 0,C 180,E1 -19310.281,E2 -19310.281} C_VEL
LIN {X 0,Y 241.994,Z 375.339,A -85,B 0,C 180,E1 -19314.489,E2 -19314.489} C_VEL
LIN {X 0,Y 241.981,Z 375.342,A -85,B 0,C 180,E1 -19318.479,E2 -19318.479} C_VEL
LIN {X 0,Y 242.015,Z 375.338,A -85,B 0,C 180,E1 -19322.312,E2 -19322.312} C_VEL
LIN {X 0,Y 242.064,Z 375.331,A -85,B 0,C 180,E1 -19326.015,E2 -19326.015} C_VEL
LIN {X 0,Y 242.115,Z 375.326,A -85,B 0,C 180,E1 -19330.939,E2 -19330.939} C_VEL
LIN {X 0,Y 242.16,Z 375.464,A -85,B 0,C 180,E1 -19331.107,E2 -19331.107} C_VEL
LIN {X 0,Y 243.676,Z 379.747,A -85,B 0,C 180,E1 -19331.607,E2 -19331.607} C_VEL
LIN {X 0,Y 247.584,Z 389.895,A -85,B 0,C 180,E1 -19333.001,E2 -19333.001} C_VEL
LIN {X 0,Y 250.658,Z 400.218,A -85,B 0,C 180,E1 -19334.579,E2 -19334.579} C_VEL
LIN {X 0,Y 251.681,Z 404.29,A -85,B 0,C 180,E1 -19335.257,E2 -19335.257} C_VEL
LIN {X 0,Y 250.352,Z 414.501,A -85,B 0,C 180,E1 -19336.814,E2 -19336.814} C_VEL
LIN {X 0,Y 248.907,Z 423.985,A -85,B 0,C 180,E1 -19338.599,E2 -19338.599} C_VEL
LIN {X 0,Y 247.411,Z 432.645,A -85,B 0,C 180,E1 -19340.598,E2 -19340.598} C_VEL
LIN {X 0,Y 245.761,Z 441.115,A -85,B 0,C 180,E1 -19343.018,E2 -19343.018} C_VEL
LIN {X 0,Y 244.585,Z 446.887,A -85,B 0,C 180,E1 -19345.054,E2 -19345.054} C_VEL
LIN {X 0,Y 243.555,Z 452.515,A -85,B 0,C 180,E1 -19347.518,E2 -19347.518} C_VEL
LIN {X 0,Y 242.704,Z 456.972,A -85,B 0,C 180,E1 -19349.999,E2 -19349.999} C_VEL
LIN {X 0,Y 242.244,Z 459.336,A -85,B 0,C 180,E1 -19351.661,E2 -19351.661} C_VEL
LIN {X 0,Y 241.93,Z 461.277,A -85,B 0,C 180,E1 -19353.33,E2 -19353.33} C_VEL
LIN {X 0,Y 241.894,Z 462.79,A -85,B 0,C 180,E1 -19354.999,E2 -19354.999} C_VEL
LIN {X 0,Y 241.875,Z 463.874,A -85,B 0,C 180,E1 -19356.673,E2 -19356.673} C_VEL
LIN {X 0,Y 242.004,Z 464.914,A -85,B 0,C 180,E1 -19360.034,E2 -19360.034} C_VEL
LIN {X 0,Y 242.284,Z 464.859,A -85,B 0,C 180,E1 -19361.714,E2 -19361.714} C_VEL
LIN {X 0,Y 243.158,Z 463.502,A -85,B 0,C 180,E1 -19365.076,E2 -19365.076} C_VEL
LIN {X 0,Y 243.821,Z 462.234,A -85,B 0,C 180,E1 -19366.752,E2 -19366.752} C_VEL
LIN {X 0,Y 244.778,Z 460.25,A -85,B 0,C 180,E1 -19368.649,E2 -19368.649} C_VEL
LIN {X 0,Y 246.616,Z 455.74,A -85,B 0,C 180,E1 -19371.743,E2 -19371.743} C_VEL
LIN {X 0,Y 248.486,Z 450.821,A -85,B 0,C 180,E1 -19374.21,E2 -19374.21} C_VEL
LIN {X 0,Y 250.703,Z 444.571,A -85,B 0,C 180,E1 -19376.648,E2 -19376.648} C_VEL
LIN {X 0,Y 253.267,Z 436.67,A -85,B 0,C 180,E1 -19379.051,E2 -19379.051} C_VEL
LIN {X 0,Y 255.577,Z 428.56,A -85,B 0,C 180,E1 -19381.036,E2 -19381.036} C_VEL
LIN {X 0,Y 258.055,Z 418.595,A -85,B 0,C 180,E1 -19383.002,E2 -19383.002} C_VEL
LIN {X 0,Y 258.418,Z 417.084,A -85,B 0,C 180,E1 -19383.252,E2 -19383.252} C_VEL
LIN {X 0,Y 256.761,Z 410.27,A -85,B 0,C 180,E1 -19384.798,E2 -19384.798} C_VEL
LIN {X 0,Y 253.627,Z 400.568,A -85,B 0,C 180,E1 -19386.857,E2 -19386.857} C_VEL
LIN {X 0,Y 249.419,Z 390.429,A -85,B 0,C 180,E1 -19388.884,E2 -19388.884} C_VEL
LIN {X 0,Y 243.616,Z 379.121,A -85,B 0,C 180,E1 -19391.066,E2 -19391.066} C_VEL
LIN {X 0,Y 242.26,Z 376.743,A -85,B 0,C 180,E1 -19391.525,E2 -19391.525} C_VEL
LIN {X 0,Y 241.93,Z 375.347,A -85,B 0,C 180,E1 -19391.714,E2 -19391.714} C_VEL
LIN {X 0,Y 241.934,Z 375.352,A -85,B 0,C 180,E1 -19395.798,E2 -19395.798} C_VEL
LIN {X 0,Y 241.986,Z 375.339,A -85,B 0,C 180,E1 -19400.286,E2 -19400.286} C_VEL
LIN {X 0,Y 242.035,Z 375.333,A -85,B 0,C 180,E1 -19404.496,E2 -19404.496} C_VEL
LIN {X 0,Y 241.972,Z 375.308,A -85,B 0,C 180,E1 -19408.479,E2 -19408.479} C_VEL
LIN {X 0,Y 242.001,Z 375.32,A -85,B 0,C 180,E1 -19412.311,E2 -19412.311} C_VEL
LIN {X 0,Y 242.055,Z 375.323,A -85,B 0,C 180,E1 -19416.015,E2 -19416.015} C_VEL
LIN {X 0,Y 242.035,Z 375.336,A -85,B 0,C 180,E1 -19419.607,E2 -19419.607} C_VEL
LIN {X 0,Y 242.16,Z 375.311,A -85,B 0,C 180,E1 -19423.277,E2 -19423.277} C_VEL
LIN {X 0,Y 242.184,Z 375.319,A -85,B 0,C 180,E1 -19428.279,E2 -19428.279} C_VEL
LIN {X 0,Y 242.432,Z 375.287,A -85,B 0,C 180,E1 -19431.665,E2 -19431.665} C_VEL
LIN {X 0,Y 242.259,Z 375.294,A -85,B 0,C 180,E1 -19435.007,E2 -19435.007} C_VEL
LIN {X 0,Y 242.636,Z 375.258,A -85,B 0,C 180,E1 -19438.34,E2 -19438.34} C_VEL
LIN {X 0,Y 242.636,Z 375.258,A -85,B 0,C 180,E1 -19441.659,E2 -19441.659} C_VEL
LIN {X 0,Y 242.43,Z 375.284,A -85,B 0,C 180,E1 -19446.659,E2 -19446.659} C_VEL
LIN {X 0,Y 242.341,Z 375.287,A -85,B 0,C 180,E1 -19450.02,E2 -19450.02} C_VEL
LIN {X 0,Y 242.162,Z 375.317,A -85,B 0,C 180,E1 -19455.141,E2 -19455.141} C_VEL
LIN {X 0,Y 242.069,Z 375.33,A -85,B 0,C 180,E1 -19458.624,E2 -19458.624} C_VEL
LIN {X 0,Y 242.009,Z 375.342,A -85,B 0,C 180,E1 -19462.18,E2 -19462.18} C_VEL
LIN {X 0,Y 242.062,Z 375.336,A -85,B 0,C 180,E1 -19465.838,E2 -19465.838} C_VEL
LIN {X 0,Y 242.006,Z 375.386,A -85,B 0,C 180,E1 -19470.665,E2 -19470.665} C_VEL
LIN {X 0,Y 243.139,Z 380.513,A -85,B 0,C 180,E1 -19475.317,E2 -19475.317} C_VEL
LIN {X 0,Y 244.125,Z 385.396,A -85,B 0,C 180,E1 -19479.297,E2 -19479.297} C_VEL
LIN {X 0,Y 245.197,Z 390.961,A -85,B 0,C 180,E1 -19483.464,E2 -19483.464} C_VEL
LIN {X 0,Y 245.416,Z 392.03,A -85,B 0,C 180,E1 -19484.227,E2 -19484.227} C_VEL
LIN {X 0,Y 245.261,Z 394.008,A -85,B 0,C 180,E1 -19485.526,E2 -19485.526} C_VEL
LIN {X 0,Y 244.263,Z 396.17,A -85,B 0,C 180,E1 -19486.799,E2 -19486.799} C_VEL
LIN {X 0,Y 239.911,Z 403.668,A -85,B 0,C 180,E1 -19491.076,E2 -19491.076} C_VEL
LIN {X 0,Y 238.204,Z 410.255,A -85,B 0,C 180,E1 -19494.995,E2 -19494.995} C_VEL
LIN {X 0,Y 238.991,Z 413.749,A -85,B 0,C 180,E1 -19495.3,E2 -19495.3} C_VEL
LIN {X 0,Y 242.232,Z 427.904,A -85,B 0,C 180,E1 -19496.81,E2 -19496.81} C_VEL
LIN {X 0,Y 244.072,Z 439.981,A -85,B 0,C 180,E1 -19498.251,E2 -19498.251} C_VEL
LIN {X 0,Y 245.121,Z 452.787,A -85,B 0,C 180,E1 -19499.987,E2 -19499.987} C_VEL
LIN {X 0,Y 245.218,Z 464.202,A -85,B 0,C 180,E1 -19501.779,E2 -19501.779} C_VEL
LIN {X 0,Y 244.535,Z 474.759,A -85,B 0,C 180,E1 -19503.7,E2 -19503.7} C_VEL
LIN {X 0,Y 243.139,Z 484.107,A -85,B 0,C 180,E1 -19505.677,E2 -19505.677} C_VEL
LIN {X 0,Y 241.296,Z 490.848,A -85,B 0,C 180,E1 -19507.3,E2 -19507.3} C_VEL
LIN {X 0,Y 238.611,Z 499.231,A -85,B 0,C 180,E1 -19509.753,E2 -19509.753} C_VEL
LIN {X 0,Y 236.669,Z 505.465,A -85,B 0,C 180,E1 -19512.03,E2 -19512.03} C_VEL
LIN {X 0,Y 235.227,Z 510.719,A -85,B 0,C 180,E1 -19514.403,E2 -19514.403} C_VEL
LIN {X 0,Y 234.118,Z 515.26,A -85,B 0,C 180,E1 -19516.99,E2 -19516.99} C_VEL
LIN {X 0,Y 233.552,Z 518.76,A -85,B 0,C 180,E1 -19519.599,E2 -19519.599} C_VEL
LIN {X 0,Y 233.501,Z 521.938,A -85,B 0,C 180,E1 -19523.086,E2 -19523.086} C_VEL
LIN {X 0,Y 233.657,Z 522.916,A -85,B 0,C 180,E1 -19524.824,E2 -19524.824} C_VEL
LIN {X 0,Y 233.984,Z 523.465,A -85,B 0,C 180,E1 -19526.557,E2 -19526.557} C_VEL
LIN {X 0,Y 234.194,Z 523.595,A -85,B 0,C 180,E1 -19528.282,E2 -19528.282} C_VEL
LIN {X 0,Y 234.325,Z 523.308,A -85,B 0,C 180,E1 -19530.001,E2 -19530.001} C_VEL
LIN {X 0,Y 234.259,Z 522.582,A -85,B 0,C 180,E1 -19531.72,E2 -19531.72} C_VEL
LIN {X 0,Y 234.142,Z 521.378,A -85,B 0,C 180,E1 -19533.443,E2 -19533.443} C_VEL
LIN {X 0,Y 233.797,Z 518.734,A -85,B 0,C 180,E1 -19536.041,E2 -19536.041} C_VEL
LIN {X 0,Y 233.637,Z 515.027,A -85,B 0,C 180,E1 -19538.652,E2 -19538.652} C_VEL
LIN {X 0,Y 233.81,Z 510.174,A -85,B 0,C 180,E1 -19541.268,E2 -19541.268} C_VEL
LIN {X 0,Y 234.65,Z 502.907,A -85,B 0,C 180,E1 -19544.307,E2 -19544.307} C_VEL
LIN {X 0,Y 235.732,Z 495.024,A -85,B 0,C 180,E1 -19546.9,E2 -19546.9} C_VEL
LIN {X 0,Y 237.344,Z 487.03,A -85,B 0,C 180,E1 -19549.011,E2 -19549.011} C_VEL
LIN {X 0,Y 238.507,Z 479.357,A -85,B 0,C 180,E1 -19550.709,E2 -19550.709} C_VEL
LIN {X 0,Y 238.898,Z 468.657,A -85,B 0,C 180,E1 -19552.714,E2 -19552.714} C_VEL
LIN {X 0,Y 239.145,Z 456.89,A -85,B 0,C 180,E1 -19554.504,E2 -19554.504} C_VEL
LIN {X 0,Y 238.884,Z 444.099,A -85,B 0,C 180,E1 -19556.071,E2 -19556.071} C_VEL
LIN {X 0,Y 237.828,Z 431.127,A -85,B 0,C 180,E1 -19557.332,E2 -19557.332} C_VEL
LIN {X 0,Y 235.995,Z 417.825,A -85,B 0,C 180,E1 -19558.346,E2 -19558.346} C_VEL
LIN {X 0,Y 235.193,Z 412.802,A -85,B 0,C 180,E1 -19558.684,E2 -19558.684} C_VEL
LIN {X 0,Y 236.753,Z 403.779,A -85,B 0,C 180,E1 -19563.78,E2 -19563.78} C_VEL
LIN {X 0,Y 237.972,Z 397.899,A -85,B 0,C 180,E1 -19567.119,E2 -19567.119} C_VEL
LIN {X 0,Y 238.347,Z 394.629,A -85,B 0,C 180,E1 -19569.059,E2 -19569.059} C_VEL
LIN {X 0,Y 237.328,Z 388.51,A -85,B 0,C 180,E1 -19572.931,E2 -19572.931} C_VEL
LIN {X 0,Y 236.238,Z 382.717,A -85,B 0,C 180,E1 -19576.824,E2 -19576.824} C_VEL
LIN {X 0,Y 234.961,Z 376.22,A -85,B 0,C 180,E1 -19581.567,E2 -19581.567} C_VEL
LIN {X 0,Y 234.935,Z 376.224,A -85,B 0,C 180,E1 -19585.363,E2 -19585.363} C_VEL
LIN {X 0,Y 234.927,Z 376.222,A -85,B 0,C 180,E1 -19589.432,E2 -19589.432} C_VEL
LIN {X 0,Y 234.999,Z 376.213,A -85,B 0,C 180,E1 -19593.795,E2 -19593.795} C_VEL
LIN {X 0,Y 235.017,Z 376.214,A -85,B 0,C 180,E1 -19598.971,E2 -19598.971} C_VEL
LIN {X 0,Y 235.102,Z 376.202,A -85,B 0,C 180,E1 -19603.06,E2 -19603.06} C_VEL
LIN {X 0,Y 235.153,Z 376.193,A -85,B 0,C 180,E1 -19607.924,E2 -19607.924} C_VEL
LIN {X 0,Y 235.397,Z 376.162,A -85,B 0,C 180,E1 -19611.415,E2 -19611.415} C_VEL
LIN {X 0,Y 235.412,Z 376.159,A -85,B 0,C 180,E1 -19613.142,E2 -19613.142} C_VEL
LIN {X 0,Y 235.602,Z 376.128,A -85,B 0,C 180,E1 -19618.291,E2 -19618.291} C_VEL
LIN {X 0,Y 235.602,Z 376.135,A -85,B 0,C 180,E1 -19621.71,E2 -19621.71} C_VEL
LIN {X 0,Y 235.412,Z 376.149,A -85,B 0,C 180,E1 -19626.859,E2 -19626.859} C_VEL
LIN {X 0,Y 235.26,Z 376.18,A -85,B 0,C 180,E1 -19630.326,E2 -19630.326} C_VEL
LIN {X 0,Y 235.12,Z 376.188,A -85,B 0,C 180,E1 -19635.606,E2 -19635.606} C_VEL
LIN {X 0,Y 235.016,Z 376.209,A -85,B 0,C 180,E1 -19639.205,E2 -19639.205} C_VEL
LIN {X 0,Y 234.968,Z 376.206,A -85,B 0,C 180,E1 -19642.883,E2 -19642.883} C_VEL
LIN {X 0,Y 234.976,Z 376.214,A -85,B 0,C 180,E1 -19646.657,E2 -19646.657} C_VEL
LIN {X 0,Y 234.938,Z 376.212,A -85,B 0,C 180,E1 -19650.567,E2 -19650.567} C_VEL
LIN {X 0,Y 234.967,Z 376.214,A -85,B 0,C 180,E1 -19654.633,E2 -19654.633} C_VEL
LIN {X 0,Y 234.948,Z 376.216,A -85,B 0,C 180,E1 -19658.944,E2 -19658.944} C_VEL
LIN {X 0,Y 234.896,Z 376.224,A -85,B 0,C 180,E1 -19663.485,E2 -19663.485} C_VEL
LIN {X 0,Y 234.896,Z 376.222,A -85,B 0,C 180,E1 -19666.514,E2 -19666.514} C_VEL
LIN {X 0,Y 234.924,Z 376.221,A -85,B 0,C 180,E1 -19671.078,E2 -19671.078} C_VEL
LIN {X 0,Y 234.936,Z 376.221,A -85,B 0,C 180,E1 -19675.362,E2 -19675.362} C_VEL
LIN {X 0,Y 234.938,Z 376.221,A -85,B 0,C 180,E1 -19679.432,E2 -19679.432} C_VEL
LIN {X 0,Y 235,Z 376.212,A -85,B 0,C 180,E1 -19683.793,E2 -19683.793} C_VEL
LIN {X 0,Y 235.017,Z 376.212,A -85,B 0,C 180,E1 -19688.969,E2 -19688.969} C_VEL
LIN {X 0,Y 235.049,Z 376.336,A -85,B 0,C 180,E1 -19690.342,E2 -19690.342} C_VEL
LIN {X 0,Y 238.635,Z 385.577,A -85,B 0,C 180,E1 -19691.562,E2 -19691.562} C_VEL
LIN {X 0,Y 241.687,Z 394.007,A -85,B 0,C 180,E1 -19692.828,E2 -19692.828} C_VEL
LIN {X 0,Y 244.717,Z 404.748,A -85,B 0,C 180,E1 -19694.608,E2 -19694.608} C_VEL
LIN {X 0,Y 244.99,Z 405.978,A -85,B 0,C 180,E1 -19694.831,E2 -19694.831} C_VEL
LIN {X 0,Y 243.371,Z 417.282,A -85,B 0,C 180,E1 -19696.642,E2 -19696.642} C_VEL
LIN {X 0,Y 241.732,Z 427.347,A -85,B 0,C 180,E1 -19698.681,E2 -19698.681} C_VEL
LIN {X 0,Y 239.922,Z 437.01,A -85,B 0,C 180,E1 -19701.152,E2 -19701.152} C_VEL
LIN {X 0,Y 238.31,Z 444.803,A -85,B 0,C 180,E1 -19703.649,E2 -19703.649} C_VEL
LIN {X 0,Y 237.215,Z 450.076,A -85,B 0,C 180,E1 -19705.751,E2 -19705.751} C_VEL
LIN {X 0,Y 236.234,Z 455.238,A -85,B 0,C 180,E1 -19708.294,E2 -19708.294} C_VEL
LIN {X 0,Y 235.425,Z 459.28,A -85,B 0,C 180,E1 -19710.854,E2 -19710.854} C_VEL
LIN {X 0,Y 234.877,Z 462.296,A -85,B 0,C 180,E1 -19713.43,E2 -19713.43} C_VEL
LIN {X 0,Y 234.856,Z 463.764,A -85,B 0,C 180,E1 -19715.149,E2 -19715.149} C_VEL
LIN {X 0,Y 234.839,Z 464.814,A -85,B 0,C 180,E1 -19716.874,E2 -19716.874} C_VEL
LIN {X 0,Y 234.994,Z 465.806,A -85,B 0,C 180,E1 -19720.336,E2 -19720.336} C_VEL
LIN {X 0,Y 235.3,Z 465.707,A -85,B 0,C 180,E1 -19722.067,E2 -19722.067} C_VEL
LIN {X 0,Y 236.263,Z 464.291,A -85,B 0,C 180,E1 -19725.527,E2 -19725.527} C_VEL
LIN {X 0,Y 237.003,Z 462.994,A -85,B 0,C 180,E1 -19727.248,E2 -19727.248} C_VEL
LIN {X 0,Y 238.354,Z 460.21,A -85,B 0,C 180,E1 -19729.819,E2 -19729.819} C_VEL
LIN {X 0,Y 239.995,Z 456.386,A -85,B 0,C 180,E1 -19732.375,E2 -19732.375} C_VEL
LIN {X 0,Y 241.958,Z 451.402,A -85,B 0,C 180,E1 -19734.907,E2 -19734.907} C_VEL
LIN {X 0,Y 244.326,Z 445.045,A -85,B 0,C 180,E1 -19737.401,E2 -19737.401} C_VEL
LIN {X 0,Y 247.011,Z 437.059,A -85,B 0,C 180,E1 -19739.861,E2 -19739.861} C_VEL
LIN {X 0,Y 249.462,Z 428.851,A -85,B 0,C 180,E1 -19741.885,E2 -19741.885} C_VEL
LIN {X 0,Y 251.987,Z 418.72,A -85,B 0,C 180,E1 -19743.903,E2 -19743.903} C_VEL
LIN {X 0,Y 249.263,Z 408.526,A -85,B 0,C 180,E1 -19746.304,E2 -19746.304} C_VEL
LIN {X 0,Y 246.14,Z 399.618,A -85,B 0,C 180,E1 -19748.26,E2 -19748.26} C_VEL
LIN {X 0,Y 241.88,Z 389.995,A -85,B 0,C 180,E1 -19750.294,E2 -19750.294} C_VEL
LIN {X 0,Y 237.097,Z 380.818,A -85,B 0,C 180,E1 -19752.178,E2 -19752.178} C_VEL
LIN {X 0,Y 235.234,Z 377.754,A -85,B 0,C 180,E1 -19752.831,E2 -19752.831} C_VEL
LIN {X 0,Y 234.883,Z 376.229,A -85,B 0,C 180,E1 -19753.055,E2 -19753.055} C_VEL
LIN {X 0,Y 234.918,Z 376.222,A -85,B 0,C 180,E1 -19756.52,E2 -19756.52} C_VEL
LIN {X 0,Y 234.953,Z 376.219,A -85,B 0,C 180,E1 -19761.085,E2 -19761.085} C_VEL
LIN {X 0,Y 234.959,Z 376.219,A -85,B 0,C 180,E1 -19765.366,E2 -19765.366} C_VEL
LIN {X 0,Y 234.92,Z 376.177,A -85,B 0,C 180,E1 -19769.43,E2 -19769.43} C_VEL
LIN {X 0,Y 234.991,Z 376.21,A -85,B 0,C 180,E1 -19773.793,E2 -19773.793} C_VEL
LIN {X 0,Y 235.009,Z 376.21,A -85,B 0,C 180,E1 -19778.969,E2 -19778.969} C_VEL
LIN {X 0,Y 235.093,Z 376.189,A -85,B 0,C 180,E1 -19783.059,E2 -19783.059} C_VEL
LIN {X 0,Y 235.144,Z 376.195,A -85,B 0,C 180,E1 -19787.923,E2 -19787.923} C_VEL
LIN {X 0,Y 235.387,Z 376.165,A -85,B 0,C 180,E1 -19791.414,E2 -19791.414} C_VEL
LIN {X 0,Y 235.403,Z 376.152,A -85,B 0,C 180,E1 -19793.141,E2 -19793.141} C_VEL
LIN {X 0,Y 235.596,Z 376.135,A -85,B 0,C 180,E1 -19798.29,E2 -19798.29} C_VEL
LIN {X 0,Y 235.596,Z 376.135,A -85,B 0,C 180,E1 -19801.709,E2 -19801.709} C_VEL
LIN {X 0,Y 235.402,Z 376.161,A -85,B 0,C 180,E1 -19806.858,E2 -19806.858} C_VEL
LIN {X 0,Y 235.249,Z 376.171,A -85,B 0,C 180,E1 -19810.326,E2 -19810.326} C_VEL
LIN {X 0,Y 235.109,Z 376.199,A -85,B 0,C 180,E1 -19815.606,E2 -19815.606} C_VEL
LIN {X 0,Y 235.005,Z 376.214,A -85,B 0,C 180,E1 -19819.206,E2 -19819.206} C_VEL
LIN {X 0,Y 234.957,Z 376.218,A -85,B 0,C 180,E1 -19822.883,E2 -19822.883} C_VEL
LIN {X 0,Y 234.966,Z 376.222,A -85,B 0,C 180,E1 -19826.658,E2 -19826.658} C_VEL
LIN {X 0,Y 235.003,Z 376.316,A -85,B 0,C 180,E1 -19829.571,E2 -19829.571} C_VEL
LIN {X 0,Y 236.061,Z 381.475,A -85,B 0,C 180,E1 -19834.448,E2 -19834.448} C_VEL
LIN {X 0,Y 237.067,Z 386.213,A -85,B 0,C 180,E1 -19838.503,E2 -19838.503} C_VEL
LIN {X 0,Y 238.114,Z 391.656,A -85,B 0,C 180,E1 -19842.754,E2 -19842.754} C_VEL
LIN {X 0,Y 238.963,Z 396.259,A -85,B 0,C 180,E1 -19846.099,E2 -19846.099} C_VEL
LIN {X 0,Y 239.905,Z 401.779,A -85,B 0,C 180,E1 -19849.874,E2 -19849.874} C_VEL
LIN {X 0,Y 239.911,Z 403.668,A -85,B 0,C 180,E1 -19851.076,E2 -19851.076} C_VEL
LIN {X 0,Y 238.978,Z 405.448,A -85,B 0,C 180,E1 -19851.948,E2 -19851.948} C_VEL
LIN {X 0,Y 237.38,Z 407.651,A -85,B 0,C 180,E1 -19852.719,E2 -19852.719} C_VEL
LIN {X 0,Y 235.136,Z 411.198,A -85,B 0,C 180,E1 -19853.603,E2 -19853.603} C_VEL
LIN {X 0,Y 233.855,Z 414.956,A -85,B 0,C 180,E1 -19854.245,E2 -19854.245} C_VEL
LIN {X 0,Y 233.833,Z 417.977,A -85,B 0,C 180,E1 -19854.599,E2 -19854.599} C_VEL
LIN {X 0,Y 236.5,Z 430.948,A -85,B 0,C 180,E1 -19856.12,E2 -19856.12} C_VEL
LIN {X 0,Y 238.089,Z 443.6,A -85,B 0,C 180,E1 -19857.769,E2 -19857.769} C_VEL
LIN {X 0,Y 238.769,Z 455.926,A -85,B 0,C 180,E1 -19859.598,E2 -19859.598} C_VEL
LIN {X 0,Y 238.539,Z 467.824,A -85,B 0,C 180,E1 -19861.636,E2 -19861.636} C_VEL
LIN {X 0,Y 237.549,Z 477.903,A -85,B 0,C 180,E1 -19863.656,E2 -19863.656} C_VEL
LIN {X 0,Y 235.765,Z 487.102,A -85,B 0,C 180,E1 -19865.804,E2 -19865.804} C_VEL
LIN {X 0,Y 232.781,Z 496.065,A -85,B 0,C 180,E1 -19868.295,E2 -19868.295} C_VEL
LIN {X 0,Y 230.421,Z 503.239,A -85,B 0,C 180,E1 -19870.825,E2 -19870.825} C_VEL
LIN {X 0,Y 228.353,Z 510.022,A -85,B 0,C 180,E1 -19873.921,E2 -19873.921} C_VEL
LIN {X 0,Y 227.169,Z 514.52,A -85,B 0,C 180,E1 -19876.585,E2 -19876.585} C_VEL
LIN {X 0,Y 226.51,Z 517.977,A -85,B 0,C 180,E1 -19879.272,E2 -19879.272} C_VEL
LIN {X 0,Y 226.426,Z 521.121,A -85,B 0,C 180,E1 -19882.869,E2 -19882.869} C_VEL
LIN {X 0,Y 226.574,Z 522.064,A -85,B 0,C 180,E1 -19884.662,E2 -19884.662} C_VEL
LIN {X 0,Y 226.904,Z 522.596,A -85,B 0,C 180,E1 -19886.45,E2 -19886.45} C_VEL
LIN {X 0,Y 227.142,Z 522.712,A -85,B 0,C 180,E1 -19888.228,E2 -19888.228} C_VEL
LIN {X 0,Y 227.278,Z 522.408,A -85,B 0,C 180,E1 -19890.001,E2 -19890.001} C_VEL
LIN {X 0,Y 227.209,Z 521.65,A -85,B 0,C 180,E1 -19891.774,E2 -19891.774} C_VEL
LIN {X 0,Y 227.061,Z 520.416,A -85,B 0,C 180,E1 -19893.55,E2 -19893.55} C_VEL
LIN {X 0,Y 226.689,Z 517.253,A -85,B 0,C 180,E1 -19896.613,E2 -19896.613} C_VEL
LIN {X 0,Y 226.589,Z 512.486,A -85,B 0,C 180,E1 -19899.823,E2 -19899.823} C_VEL
LIN {X 0,Y 227.129,Z 506.165,A -85,B 0,C 180,E1 -19902.965,E2 -19902.965} C_VEL
LIN {X 0,Y 228.007,Z 499.266,A -85,B 0,C 180,E1 -19905.648,E2 -19905.648} C_VEL
LIN {X 0,Y 229.187,Z 492.272,A -85,B 0,C 180,E1 -19907.859,E2 -19907.859} C_VEL
LIN {X 0,Y 230.904,Z 483.898,A -85,B 0,C 180,E1 -19910.025,E2 -19910.025} C_VEL
LIN {X 0,Y 231.677,Z 476.826,A -85,B 0,C 180,E1 -19911.582,E2 -19911.582} C_VEL
LIN {X 0,Y 232.062,Z 466.105,A -85,B 0,C 180,E1 -19913.596,E2 -19913.596} C_VEL
LIN {X 0,Y 232.326,Z 455.003,A -85,B 0,C 180,E1 -19915.297,E2 -19915.297} C_VEL
LIN {X 0,Y 232.06,Z 443.197,A -85,B 0,C 180,E1 -19916.777,E2 -19916.777} C_VEL
LIN {X 0,Y 231.013,Z 430.194,A -85,B 0,C 180,E1 -19918.085,E2 -19918.085} C_VEL
LIN {X 0,Y 229.128,Z 416.998,A -85,B 0,C 180,E1 -19919.139,E2 -19919.139} C_VEL
LIN {X 0,Y 228.337,Z 411.893,A -85,B 0,C 180,E1 -19919.504,E2 -19919.504} C_VEL
LIN {X 0,Y 229.853,Z 403.606,A -85,B 0,C 180,E1 -19924.355,E2 -19924.355} C_VEL
LIN {X 0,Y 231.069,Z 397.887,A -85,B 0,C 180,E1 -19927.74,E2 -19927.74} C_VEL
LIN {X 0,Y 231.211,Z 394.746,A -85,B 0,C 180,E1 -19929.669,E2 -19929.669} C_VEL
LIN {X 0,Y 230.356,Z 389.803,A -85,B 0,C 180,E1 -19932.927,E2 -19932.927} C_VEL
LIN {X 0,Y 229.073,Z 383.155,A -85,B 0,C 180,E1 -19937.549,E2 -19937.549} C_VEL
LIN {X 0,Y 227.934,Z 377.096,A -85,B 0,C 180,E1 -19942.121,E2 -19942.121} C_VEL
LIN {X 0,Y 227.884,Z 377.101,A -85,B 0,C 180,E1 -19946.378,E2 -19946.378} C_VEL
LIN {X 0,Y 227.909,Z 377.096,A -85,B 0,C 180,E1 -19950.437,E2 -19950.437} C_VEL
LIN {X 0,Y 227.933,Z 377.095,A -85,B 0,C 180,E1 -19954.427,E2 -19954.427} C_VEL
LIN {X 0,Y 227.968,Z 377.092,A -85,B 0,C 180,E1 -19958.288,E2 -19958.288} C_VEL
LIN {X 0,Y 228.04,Z 377.083,A -85,B 0,C 180,E1 -19962.826,E2 -19962.826} C_VEL
LIN {X 0,Y 228.1,Z 377.071,A -85,B 0,C 180,E1 -19967.545,E2 -19967.545} C_VEL
LIN {X 0,Y 228.331,Z 377.042,A -85,B 0,C 180,E1 -19971.147,E2 -19971.147} C_VEL
LIN {X 0,Y 228.364,Z 377.038,A -85,B 0,C 180,E1 -19972.929,E2 -19972.929} C_VEL
LIN {X 0,Y 228.56,Z 377.005,A -85,B 0,C 180,E1 -19978.238,E2 -19978.238} C_VEL
LIN {X 0,Y 228.561,Z 377.012,A -85,B 0,C 180,E1 -19981.762,E2 -19981.762} C_VEL
LIN {X 0,Y 228.365,Z 377.026,A -85,B 0,C 180,E1 -19987.072,E2 -19987.072} C_VEL
LIN {X 0,Y 228.178,Z 377.06,A -85,B 0,C 180,E1 -19990.65,E2 -19990.65} C_VEL
LIN {X 0,Y 228.064,Z 377.069,A -85,B 0,C 180,E1 -19996.102,E2 -19996.102} C_VEL
LIN {X 0,Y 227.95,Z 377.091,A -85,B 0,C 180,E1 -19999.825,E2 -19999.825} C_VEL
LIN {X 0,Y 227.921,Z 377.086,A -85,B 0,C 180,E1 -20003.632,E2 -20003.632} C_VEL
LIN {X 0,Y 227.892,Z 377.099,A -85,B 0,C 180,E1 -20007.555,E2 -20007.555} C_VEL
LIN {X 0,Y 227.879,Z 377.095,A -85,B 0,C 180,E1 -20011.622,E2 -20011.622} C_VEL
LIN {X 0,Y 227.906,Z 377.096,A -85,B 0,C 180,E1 -20015.868,E2 -20015.868} C_VEL
LIN {X 0,Y 227.84,Z 377.102,A -85,B 0,C 180,E1 -20020.375,E2 -20020.375} C_VEL
LIN {X 0,Y 227.841,Z 377.102,A -85,B 0,C 180,E1 -20025.192,E2 -20025.192} C_VEL
LIN {X 0,Y 227.832,Z 377.102,A -85,B 0,C 180,E1 -20029.623,E2 -20029.623} C_VEL
